C01788=1016.135,48.683,-123.582,-24.251,21.472,-42.282
C01789=1016.137,48.283,-123.546,-24.251,21.474,-42.286
C01790=1016.140,47.883,-123.510,-24.251,21.474,-42.290
C01791=1016.142,47.483,-123.475,-24.250,21.474,-42.295
C01792=1016.145,47.083,-123.439,-24.249,21.475,-42.299
C01793=1016.149,46.682,-123.404,-24.249,21.475,-42.302
C01794=1016.151,46.283,-123.368,-24.248,21.475,-42.308
C01795=1016.153,45.882,-123.332,-24.247,21.475,-42.311
C01796=1016.156,45.482,-123.297,-24.247,21.477,-42.316
C01797=1016.158,45.082,-123.261,-24.246,21.477,-42.321
C01798=1016.161,44.683,-123.225,-24.246,21.477,-42.325
C01799=1016.163,44.282,-123.190,-24.245,21.477,-42.330
C01800=1016.166,43.882,-123.154,-24.244,21.477,-42.333
C01801=1016.169,43.482,-123.119,-24.244,21.479,-42.338
C01802=1016.171,43.082,-123.084,-24.243,21.479,-42.343
C01803=1016.174,42.683,-123.048,-24.243,21.479,-42.347
C01804=1016.177,42.282,-123.012,-24.242,21.479,-42.352
C01805=1016.179,41.882,-122.977,-24.241,21.479,-42.356
C01806=1016.181,41.482,-122.941,-24.241,21.480,-42.359
C01807=1016.184,41.082,-122.906,-24.240,21.481,-42.365
C01808=1016.186,40.683,-122.871,-24.240,21.481,-42.369
C01809=1016.188,40.283,-122.835,-24.239,21.481,-42.374
C01810=1016.191,39.882,-122.800,-24.238,21.481,-42.378
C01811=1016.194,39.483,-122.764,-24.238,21.482,-42.383
C01812=1016.196,39.083,-122.728,-24.237,21.483,-42.387
C01813=1016.199,38.683,-122.694,-24.237,21.483,-42.391
C01814=1016.201,38.283,-122.658,-24.236,21.483,-42.396
C01815=1016.203,37.882,-122.623,-24.235,21.483,-42.400
C01816=1016.205,37.483,-122.587,-24.235,21.484,-42.405
C01817=1016.207,37.084,-122.553,-24.234,21.485,-42.409
C01818=1016.209,36.684,-122.518,-24.233,21.484,-42.414
C01819=1016.212,36.284,-122.482,-24.233,21.485,-42.418
C01820=1016.214,35.884,-122.447,-24.232,21.486,-42.424
C01821=1016.216,35.484,-122.411,-24.231,21.486,-42.428
C01822=1016.219,35.084,-122.376,-24.231,21.486,-42.433
C01823=1016.220,34.685,-122.341,-24.230,21.486,-42.437
C01824=1016.222,34.285,-122.305,-24.229,21.487,-42.442
C01825=1016.225,33.885,-122.271,-24.229,21.488,-42.446
C01826=1016.227,33.486,-122.236,-24.228,21.487,-42.451
C01827=1016.229,33.086,-122.200,-24.228,21.489,-42.455
C01828=1016.232,32.686,-122.165,-24.227,21.489,-42.461
C01829=1016.233,32.287,-122.130,-24.226,21.489,-42.464
C01830=1016.235,31.887,-122.095,-24.226,21.489,-42.469
C01831=1016.237,31.487,-122.060,-24.225,21.490,-42.474
C01832=1016.239,31.087,-122.025,-24.224,21.490,-42.479
C01833=1016.241,30.688,-121.990,-24.224,21.491,-42.483
C01834=1016.243,30.289,-121.954,-24.223,21.491,-42.488
C01835=1016.245,29.889,-121.920,-24.223,21.492,-42.492
C01836=1016.247,29.490,-121.885,-24.222,21.492,-42.497
C01837=1016.249,29.090,-121.850,-24.221,21.492,-42.501
C01838=1016.250,28.691,-121.815,-24.221,21.493,-42.507
C01839=1016.252,28.291,-121.781,-24.220,21.493,-42.510
C01840=1016.255,27.891,-121.745,-24.219,21.493,-42.516
C01841=1016.256,27.492,-121.710,-24.219,21.495,-42.520
C01842=1016.258,27.093,-121.675,-24.218,21.494,-42.525
C01843=1016.260,26.693,-121.641,-24.218,21.495,-42.529
C01844=1016.261,26.294,-121.606,-24.217,21.496,-42.534
C01845=1016.263,25.895,-121.571,-24.216,21.496,-42.540
C01846=1016.265,25.495,-121.536,-24.215,21.496,-42.543
C01847=1016.267,25.096,-121.501,-24.215,21.497,-42.549
C01848=1016.269,24.697,-121.467,-24.214,21.497,-42.553
C01849=1016.271,24.298,-121.432,-24.213,21.497,-42.558
C01850=1016.272,23.915,-121.398,-24.213,21.498,-42.562
C01851=1016.273,23.584,-121.370,-24.213,21.498,-42.564
C01852=1016.275,23.313,-121.346,-24.212,21.498,-42.567
C01853=1016.275,23.078,-121.326,-24.211,21.499,-42.573
C01854=1016.277,22.846,-121.305,-24.211,21.500,-42.577
C01855=1016.278,22.580,-121.283,-24.211,21.500,-42.580
C01856=1016.278,22.258,-121.254,-24.210,21.500,-42.584
C01857=1016.280,21.883,-121.222,-24.210,21.501,-42.586
C01858=1016.282,21.470,-121.186,-24.209,21.501,-42.593
C01859=1016.283,21.225,-121.165,-24.208,21.501,-42.597
C01860=1016.284,20.953,-121.142,-24.208,21.502,-42.599
C01861=1016.285,20.662,-121.116,-24.207,21.501,-42.602
C01862=1016.286,20.365,-121.090,-24.207,21.501,-42.604
C01863=1016.288,20.078,-121.065,-24.207,21.503,-42.606
C01864=1016.288,19.812,-121.042,-24.206,21.502,-42.610
C01865=1016.289,19.575,-121.022,-24.206,21.503,-42.613
C01866=1016.290,19.364,-121.004,-24.205,21.503,-42.617
C01867=1016.291,18.968,-120.970,-24.205,21.503,-42.622
C01868=1016.293,18.571,-120.935,-24.204,21.503,-42.626
C01869=1016.294,18.175,-120.901,-24.203,21.504,-42.632
C01870=1016.296,17.780,-120.867,-24.203,21.505,-42.635
C01871=1016.297,17.386,-120.832,-24.202,21.505,-42.641
C01872=1016.298,16.993,-120.799,-24.201,21.505,-42.646
C01873=1016.299,16.600,-120.765,-24.201,21.506,-42.650
C01874=1016.301,16.208,-120.731,-24.200,21.506,-42.656
C01875=1016.302,15.816,-120.697,-24.200,21.507,-42.659
C01876=1016.304,15.427,-120.664,-24.199,21.507,-42.665
C01877=1016.305,15.037,-120.630,-24.198,21.508,-42.670
C01878=1016.306,14.649,-120.597,-24.198,21.508,-42.674
C01879=1016.307,14.260,-120.563,-24.197,21.509,-42.680
C01880=1016.309,13.873,-120.530,-24.196,21.509,-42.683
C01881=1016.310,13.485,-120.497,-24.196,21.509,-42.689
C01882=1016.311,13.098,-120.463,-24.195,21.511,-42.693
C01883=1016.312,12.712,-120.430,-24.194,21.510,-42.698
C01884=1016.313,12.325,-120.397,-24.193,21.510,-42.703
C01885=1016.314,11.939,-120.364,-24.193,21.512,-42.707
C01886=1016.315,11.552,-120.330,-24.192,21.511,-42.713
C01887=1016.317,11.167,-120.298,-24.192,21.512,-42.716
C01888=1016.317,10.784,-120.265,-24.191,21.513,-42.722
C01889=1016.319,10.403,-120.232,-24.191,21.513,-42.726
C01890=1016.320,10.025,-120.201,-24.190,21.513,-42.731
C01891=1016.320,9.648,-120.168,-24.189,21.514,-42.737
C01892=1016.321,9.273,-120.136,-24.189,21.514,-42.740
C01893=1016.323,8.896,-120.104,-24.188,21.515,-42.746
C01894=1016.323,8.518,-120.071,-24.187,21.515,-42.751
C01895=1016.324,8.138,-120.039,-24.187,21.516,-42.755
C01896=1016.325,7.753,-120.006,-24.186,21.516,-42.761
C01897=1016.327,7.366,-119.973,-24.185,21.517,-42.764
C01898=1016.326,6.975,-119.940,-24.185,21.517,-42.770
C01899=1016.328,6.583,-119.906,-24.184,21.517,-42.775
C01900=1016.329,6.190,-119.873,-24.183,21.519,-42.779
C01901=1016.329,5.797,-119.840,-24.182,21.518,-42.785
C01902=1016.331,5.401,-119.806,-24.182,21.519,-42.790
C01903=1016.331,5.006,-119.772,-24.181,21.520,-42.794
C01904=1016.332,4.612,-119.739,-24.180,21.519,-42.799
C01905=1016.333,4.215,-119.705,-24.180,21.520,-42.805
C01906=1016.333,3.826,-119.672,-24.179,21.521,-42.809
C01907=1016.334,3.467,-119.641,-24.179,21.521,-42.812
C01908=1016.335,3.139,-119.613,-24.178,21.521,-42.817
C01909=1016.335,2.825,-119.586,-24.177,21.522,-42.823
C01910=1016.336,2.503,-119.560,-24.177,21.522,-42.827
C01911=1016.337,2.150,-119.530,-24.176,21.523,-42.833
C01912=1016.337,1.764,-119.496,-24.175,21.524,-42.836
C01913=1016.338,1.367,-119.463,-24.175,21.523,-42.841
C01914=1016.338,0.967,-119.430,-24.174,21.525,-42.846
C01915=1016.339,0.567,-119.396,-24.173,21.525,-42.851
C01916=1016.340,0.166,-119.361,-24.173,21.525,-42.857
C01917=1016.340,-0.237,-119.327,-24.172,21.525,-42.862
C01918=1016.341,-0.644,-119.293,-24.171,21.526,-42.867
C01919=1016.341,-1.051,-119.259,-24.171,21.527,-42.872
C01920=1016.342,-1.462,-119.224,-24.170,21.527,-42.877
C01921=1016.342,-1.874,-119.190,-24.169,21.528,-42.882
C01922=1016.343,-2.289,-119.155,-24.169,21.529,-42.888
C01923=1016.343,-2.705,-119.120,-24.168,21.529,-42.893
C01924=1016.344,-3.125,-119.084,-24.167,21.529,-42.899
C01925=1016.345,-3.547,-119.049,-24.166,21.530,-42.904
C01926=1016.345,-3.758,-119.031,-24.166,21.530,-42.908
C01927=1016.345,-3.970,-119.013,-24.165,21.530,-42.910
C01928=1016.345,-4.184,-118.995,-24.165,21.530,-42.913
C01929=1016.345,-4.400,-118.977,-24.165,21.531,-42.915
C01930=1016.346,-4.616,-118.959,-24.164,21.531,-42.919
C01931=1016.347,-4.834,-118.941,-24.164,21.531,-42.921
C01932=1016.346,-5.054,-118.922,-24.163,21.532,-42.925
C01933=1016.346,-5.276,-118.903,-24.163,21.532,-42.927
C01934=1016.347,-5.499,-118.885,-24.163,21.532,-42.930
C01935=1016.347,-5.722,-118.866,-24.162,21.532,-42.934
C01936=1016.347,-5.946,-118.847,-24.162,21.533,-42.935
C01937=1016.347,-6.171,-118.828,-24.161,21.533,-42.939
C01938=1016.347,-6.394,-118.809,-24.161,21.533,-42.941
C01939=1016.347,-6.618,-118.791,-24.161,21.533,-42.944
C01940=1016.348,-6.842,-118.772,-24.160,21.534,-42.947
C01941=1016.348,-7.064,-118.754,-24.160,21.534,-42.950
C01942=1016.348,-7.285,-118.735,-24.160,21.535,-42.952
C01943=1016.348,-7.506,-118.716,-24.159,21.534,-42.956
C01944=1016.348,-7.725,-118.699,-24.159,21.535,-42.959
C01945=1016.349,-7.943,-118.680,-24.158,21.535,-42.961
C01946=1016.348,-8.160,-118.662,-24.158,21.536,-42.965
C01947=1016.349,-8.377,-118.644,-24.158,21.536,-42.967
C01948=1016.349,-8.594,-118.626,-24.157,21.536,-42.971
C01949=1016.348,-8.810,-118.607,-24.157,21.537,-42.973
C01950=1016.348,-9.027,-118.589,-24.156,21.536,-42.976
C01951=1016.349,-9.243,-118.572,-24.156,21.537,-42.980
C01952=1016.349,-9.460,-118.553,-24.156,21.537,-42.982
C01953=1016.349,-9.676,-118.535,-24.155,21.538,-42.985
C01954=1016.349,-9.893,-118.517,-24.155,21.538,-42.987
C01955=1016.349,-10.108,-118.499,-24.154,21.538,-42.991
C01956=1016.349,-10.324,-118.482,-24.154,21.539,-42.993
C01957=1016.349,-10.539,-118.463,-24.154,21.538,-42.996
C01958=1016.350,-10.754,-118.445,-24.153,21.539,-42.998
C01959=1016.349,-10.969,-118.428,-24.153,21.539,-43.002
C01960=1016.349,-11.183,-118.410,-24.152,21.539,-43.006
C01961=1016.349,-11.396,-118.392,-24.152,21.540,-43.007
C01962=1016.349,-11.610,-118.374,-24.152,21.540,-43.011
C01963=1016.350,-11.822,-118.357,-24.151,21.540,-43.013
C01964=1016.350,-12.035,-118.339,-24.151,21.540,-43.016
C01965=1016.350,-12.247,-118.321,-24.151,21.541,-43.019
C01966=1016.349,-12.458,-118.304,-24.150,21.541,-43.022
C01967=1016.349,-12.670,-118.286,-24.150,21.542,-43.024
C01968=1016.349,-13.089,-118.252,-24.149,21.542,-43.029
C01969=1016.349,-13.506,-118.216,-24.148,21.543,-43.035
C01970=1016.349,-13.921,-118.182,-24.148,21.543,-43.041
C01971=1016.349,-14.332,-118.149,-24.147,21.544,-43.046
C01972=1016.349,-14.741,-118.115,-24.146,21.544,-43.052
C01973=1016.349,-15.146,-118.081,-24.145,21.545,-43.057
C01974=1016.349,-15.549,-118.048,-24.145,21.545,-43.063
C01975=1016.349,-15.950,-118.015,-24.144,21.546,-43.068
C01976=1016.349,-16.349,-117.982,-24.143,21.546,-43.074
C01977=1016.348,-16.748,-117.948,-24.142,21.547,-43.079
C01978=1016.348,-17.146,-117.915,-24.142,21.548,-43.085
C01979=1016.348,-17.544,-117.883,-24.141,21.547,-43.090
C01980=1016.348,-17.955,-117.849,-24.140,21.548,-43.098
C01981=1016.347,-18.203,-117.829,-24.139,21.549,-43.101
C01982=1016.347,-18.490,-117.804,-24.139,21.549,-43.105
C01983=1016.347,-18.802,-117.779,-24.139,21.550,-43.107
C01984=1016.347,-19.113,-117.753,-24.139,21.550,-43.109
C01985=1016.347,-19.401,-117.730,-24.138,21.550,-43.113
C01986=1016.347,-19.651,-117.709,-24.138,21.551,-43.116
C01987=1016.346,-20.061,-117.675,-24.136,21.551,-43.123
C01988=1016.346,-20.459,-117.643,-24.136,21.552,-43.129
C01989=1016.345,-20.857,-117.609,-24.135,21.553,-43.135
C01990=1016.345,-21.254,-117.577,-24.134,21.552,-43.140
C01991=1016.345,-21.652,-117.544,-24.134,21.553,-43.146
C01992=1016.344,-22.049,-117.512,-24.133,21.554,-43.151
C01993=1016.344,-22.447,-117.479,-24.132,21.554,-43.156
C01994=1016.343,-22.844,-117.447,-24.131,21.555,-43.162
C01995=1016.342,-23.242,-117.414,-24.131,21.555,-43.168
C01996=1016.342,-23.639,-117.382,-24.130,21.556,-43.173
C01997=1016.342,-24.037,-117.349,-24.129,21.556,-43.178
C01998=1016.341,-24.434,-117.317,-24.128,21.557,-43.184
C01999=1016.341,-24.832,-117.284,-24.128,21.558,-43.190
C02000=1016.340,-25.229,-117.252,-24.127,21.558,-43.195
C02001=1016.339,-25.627,-117.219,-24.126,21.558,-43.201
C02002=1016.339,-26.024,-117.187,-24.125,21.559,-43.206
C02003=1016.338,-26.422,-117.154,-24.125,21.560,-43.212
C02004=1016.337,-26.819,-117.122,-24.124,21.560,-43.217
C02005=1016.336,-27.216,-117.090,-24.123,21.561,-43.221
C02006=1016.336,-27.614,-117.057,-24.123,21.562,-43.227
C02007=1016.335,-28.012,-117.025,-24.122,21.562,-43.232
C02008=1016.334,-28.410,-116.993,-24.121,21.562,-43.238
C02009=1016.334,-28.807,-116.961,-24.120,21.563,-43.243
C02010=1016.333,-29.204,-116.929,-24.120,21.564,-43.249
C02011=1016.331,-29.602,-116.896,-24.119,21.565,-43.255
C02012=1016.331,-29.999,-116.864,-24.118,21.565,-43.260
C02013=1016.330,-30.397,-116.832,-24.117,21.565,-43.265
C02014=1016.329,-30.794,-116.800,-24.117,21.566,-43.271
C02015=1016.328,-31.191,-116.768,-24.116,21.567,-43.277
C02016=1016.327,-31.589,-116.735,-24.115,21.568,-43.282
C02017=1016.326,-31.986,-116.703,-24.114,21.567,-43.287
C02018=1016.325,-32.383,-116.671,-24.114,21.568,-43.293
C02019=1016.325,-32.781,-116.639,-24.113,21.569,-43.299
C02020=1016.323,-33.179,-116.607,-24.112,21.570,-43.304
C02021=1016.322,-33.576,-116.575,-24.111,21.570,-43.310
C02022=1016.321,-33.973,-116.543,-24.111,21.570,-43.315
C02023=1016.321,-34.371,-116.511,-24.110,21.571,-43.321
C02024=1016.319,-34.768,-116.479,-24.109,21.571,-43.328
C02025=1016.318,-35.166,-116.447,-24.108,21.572,-43.334
C02026=1016.317,-35.563,-116.414,-24.107,21.572,-43.339
C02027=1016.315,-35.960,-116.383,-24.107,21.573,-43.344
C02028=1016.315,-36.357,-116.351,-24.106,21.573,-43.350
C02029=1016.313,-36.755,-116.319,-24.105,21.574,-43.356
C02030=1016.312,-37.152,-116.287,-24.105,21.575,-43.361
C02031=1016.311,-37.549,-116.256,-24.104,21.575,-43.366
C02032=1016.310,-37.947,-116.223,-24.103,21.576,-43.372
C02033=1016.308,-38.344,-116.192,-24.102,21.576,-43.378
C02034=1016.307,-38.741,-116.159,-24.102,21.577,-43.383
C02035=1016.305,-39.138,-116.128,-24.101,21.578,-43.389
C02036=1016.304,-39.536,-116.097,-24.100,21.578,-43.394
C02037=1016.303,-39.934,-116.064,-24.099,21.579,-43.400
C02038=1016.301,-40.331,-116.033,-24.099,21.579,-43.405
C02039=1016.300,-40.728,-116.001,-24.098,21.580,-43.411
C02040=1016.298,-41.126,-115.969,-24.097,21.581,-43.417
C02041=1016.297,-41.523,-115.937,-24.096,21.582,-43.422
C02042=1016.296,-41.920,-115.906,-24.096,21.582,-43.427
C02043=1016.294,-42.317,-115.875,-24.095,21.582,-43.433
C02044=1016.292,-42.715,-115.843,-24.094,21.583,-43.439
C02045=1016.291,-43.112,-115.811,-24.093,21.584,-43.444
C02046=1016.289,-43.509,-115.779,-24.092,21.584,-43.451
C02047=1016.288,-43.906,-115.749,-24.092,21.585,-43.457
C02048=1016.286,-44.304,-115.717,-24.091,21.585,-43.462
C02049=1016.284,-44.701,-115.685,-24.090,21.585,-43.468
C02050=1016.283,-45.098,-115.653,-24.089,21.586,-43.473
C02051=1016.281,-45.495,-115.622,-24.089,21.587,-43.479
C02052=1016.279,-45.892,-115.590,-24.088,21.588,-43.485
C02053=1016.278,-46.290,-115.559,-24.087,21.589,-43.490
C02054=1016.276,-46.687,-115.527,-24.086,21.588,-43.496
C02055=1016.274,-47.083,-115.496,-24.086,21.589,-43.501
C02056=1016.272,-47.481,-115.464,-24.085,21.590,-43.507
C02057=1016.271,-47.878,-115.433,-24.084,21.591,-43.512
C02058=1016.269,-48.275,-115.402,-24.084,21.592,-43.518
C02059=1016.267,-48.673,-115.371,-24.083,21.592,-43.525
C02060=1016.265,-49.070,-115.339,-24.082,21.592,-43.531
C02061=1016.263,-49.466,-115.308,-24.081,21.592,-43.536
C02062=1016.261,-49.863,-115.276,-24.080,21.593,-43.542
C02063=1016.259,-50.261,-115.244,-24.080,21.594,-43.547
C02064=1016.257,-50.658,-115.214,-24.079,21.595,-43.553
C02065=1016.255,-51.055,-115.183,-24.078,21.595,-43.558
C02066=1016.253,-51.452,-115.152,-24.077,21.596,-43.564
C02067=1016.251,-51.848,-115.121,-24.077,21.597,-43.570
C02068=1016.249,-52.246,-115.089,-24.076,21.598,-43.575
C02069=1016.247,-52.642,-115.058,-24.075,21.598,-43.581
C02070=1016.245,-53.039,-115.027,-24.074,21.598,-43.588
C02071=1016.242,-53.436,-114.996,-24.073,21.599,-43.593
C02072=1016.241,-53.833,-114.965,-24.073,21.599,-43.599
C02073=1016.238,-54.231,-114.933,-24.072,21.600,-43.604
C02074=1016.236,-54.627,-114.902,-24.071,21.601,-43.610
C02075=1016.234,-55.024,-114.871,-24.071,21.602,-43.616
C02076=1016.231,-55.421,-114.840,-24.070,21.603,-43.621
C02077=1016.230,-55.819,-114.809,-24.069,21.602,-43.627
C02078=1016.227,-56.216,-114.778,-24.068,21.603,-43.632
C02079=1016.224,-56.614,-114.747,-24.067,21.603,-43.639
C02080=1016.223,-57.012,-114.716,-24.067,21.604,-43.645
C02081=1016.220,-57.410,-114.685,-24.066,21.605,-43.651
C02082=1016.218,-57.809,-114.654,-24.065,21.606,-43.656
C02083=1016.215,-58.208,-114.623,-24.064,21.606,-43.662
C02084=1016.212,-58.607,-114.592,-24.064,21.607,-43.667
C02085=1016.210,-59.008,-114.561,-24.063,21.608,-43.673
C02086=1016.208,-59.409,-114.529,-24.062,21.608,-43.680
C02087=1016.205,-59.811,-114.499,-24.061,21.609,-43.686
C02088=1016.202,-60.212,-114.468,-24.061,21.610,-43.691
C02089=1016.200,-60.614,-114.436,-24.060,21.610,-43.697
C02090=1016.197,-61.018,-114.405,-24.059,21.610,-43.702
C02091=1016.195,-61.421,-114.374,-24.058,21.611,-43.708
C02092=1016.192,-61.825,-114.342,-24.057,21.611,-43.715
C02093=1016.190,-62.230,-114.311,-24.057,21.612,-43.720
C02094=1016.186,-62.635,-114.280,-24.056,21.613,-43.726
C02095=1016.183,-63.041,-114.248,-24.055,21.614,-43.732
C02096=1016.181,-63.447,-114.217,-24.054,21.615,-43.737
C02097=1016.178,-63.854,-114.185,-24.053,21.615,-43.744
C02098=1016.175,-64.261,-114.154,-24.053,21.615,-43.750
C02099=1016.171,-64.669,-114.122,-24.052,21.616,-43.756
C02100=1016.170,-65.077,-114.091,-24.051,21.617,-43.761
C02101=1016.166,-65.486,-114.060,-24.050,21.617,-43.768
C02102=1016.163,-65.895,-114.028,-24.049,21.618,-43.774
C02103=1016.161,-66.303,-113.996,-24.049,21.619,-43.780
C02104=1016.157,-66.713,-113.965,-24.048,21.620,-43.785
C02105=1016.154,-67.122,-113.933,-24.047,21.620,-43.791
C02106=1016.151,-67.533,-113.902,-24.046,21.621,-43.798
C02107=1016.148,-67.943,-113.870,-24.046,21.621,-43.804
C02108=1016.144,-68.354,-113.839,-24.045,21.622,-43.809
C02109=1016.141,-68.764,-113.807,-24.044,21.623,-43.815
C02110=1016.138,-69.175,-113.776,-24.043,21.623,-43.822
C02111=1016.135,-69.585,-113.744,-24.042,21.624,-43.827
C02112=1016.131,-69.997,-113.713,-24.042,21.625,-43.833
C02113=1016.128,-70.407,-113.681,-24.041,21.625,-43.839
C02114=1016.125,-70.818,-113.650,-24.040,21.626,-43.846
C02115=1016.122,-71.229,-113.619,-24.039,21.626,-43.851
C02116=1016.118,-71.640,-113.587,-24.039,21.627,-43.857
C02117=1016.115,-72.052,-113.556,-24.038,21.628,-43.865
C02118=1016.112,-72.462,-113.524,-24.037,21.629,-43.870
C02119=1016.107,-72.873,-113.493,-24.036,21.630,-43.876
C02120=1016.104,-73.283,-113.462,-24.035,21.631,-43.881
C02121=1016.101,-73.695,-113.431,-24.034,21.631,-43.888
C02122=1016.097,-74.105,-113.399,-24.034,21.632,-43.894
C02123=1016.093,-74.516,-113.368,-24.033,21.632,-43.900
C02124=1016.089,-74.926,-113.337,-24.032,21.633,-43.905
C02125=1016.086,-75.336,-113.305,-24.031,21.633,-43.912
C02126=1016.083,-75.746,-113.275,-24.031,21.634,-43.918
C02127=1016.078,-76.156,-113.243,-24.030,21.635,-43.924
C02128=1016.075,-76.565,-113.212,-24.029,21.636,-43.929
C02129=1016.071,-76.974,-113.181,-24.028,21.636,-43.936
C02130=1016.068,-77.383,-113.150,-24.027,21.637,-43.942
C02131=1016.064,-77.791,-113.119,-24.027,21.637,-43.948
C02132=1016.060,-78.199,-113.088,-24.026,21.638,-43.953
C02133=1016.056,-78.607,-113.057,-24.025,21.638,-43.960
C02134=1016.052,-79.014,-113.026,-24.024,21.639,-43.966
C02135=1016.048,-79.421,-112.995,-24.023,21.640,-43.972
C02136=1016.044,-79.826,-112.965,-24.023,21.641,-43.977
C02137=1016.040,-80.233,-112.934,-24.022,21.641,-43.984
C02138=1016.036,-80.638,-112.904,-24.021,21.642,-43.990
C02139=1016.032,-81.042,-112.873,-24.020,21.643,-43.995
C02140=1016.028,-81.446,-112.843,-24.020,21.643,-44.001
C02141=1016.024,-81.850,-112.812,-24.019,21.644,-44.007
C02142=1016.020,-82.252,-112.782,-24.018,21.644,-44.014
C02143=1016.016,-82.654,-112.752,-24.017,21.645,-44.019
C02144=1016.012,-83.056,-112.721,-24.016,21.646,-44.025
C02145=1016.008,-83.457,-112.692,-24.016,21.647,-44.031
C02146=1016.003,-83.857,-112.661,-24.015,21.648,-44.036
C02147=1015.999,-84.257,-112.631,-24.014,21.648,-44.043
C02148=1015.995,-84.663,-112.600,-24.013,21.649,-44.049
C02149=1015.992,-84.887,-112.584,-24.013,21.649,-44.053
C02150=1015.989,-85.128,-112.566,-24.012,21.650,-44.056
C02151=1015.988,-85.381,-112.547,-24.012,21.649,-44.060
C02152=1015.984,-85.636,-112.528,-24.012,21.650,-44.062
C02153=1015.981,-85.882,-112.509,-24.011,21.650,-44.065
C02154=1015.979,-86.111,-112.492,-24.011,21.651,-44.069
C02155=1015.974,-86.522,-112.461,-24.010,21.652,-44.077
C02156=1015.970,-86.909,-112.432,-24.009,21.652,-44.082
C02157=1015.967,-87.289,-112.403,-24.008,21.652,-44.087
C02158=1015.962,-87.661,-112.375,-24.007,21.653,-44.093
C02159=1015.958,-88.033,-112.347,-24.007,21.654,-44.099
C02160=1015.953,-88.409,-112.320,-24.006,21.655,-44.104
C02161=1015.949,-88.816,-112.289,-24.005,21.656,-44.112
C02162=1015.946,-89.063,-112.271,-24.005,21.656,-44.116
C02163=1015.943,-89.339,-112.250,-24.004,21.657,-44.117
C02164=1015.940,-89.623,-112.229,-24.004,21.656,-44.121
C02165=1015.936,-89.897,-112.209,-24.003,21.657,-44.124
C02166=1015.933,-90.148,-112.190,-24.003,21.657,-44.128
C02167=1015.931,-90.366,-112.173,-24.002,21.658,-44.132
C02168=1015.926,-90.762,-112.144,-24.002,21.659,-44.138
C02169=1015.921,-91.156,-112.115,-24.001,21.659,-44.145
C02170=1015.917,-91.548,-112.086,-24.000,21.660,-44.150
C02171=1015.912,-91.941,-112.056,-23.999,21.660,-44.156
C02172=1015.908,-92.332,-112.027,-23.999,21.661,-44.162
C02173=1015.903,-92.723,-111.998,-23.998,21.662,-44.167
C02174=1015.898,-93.113,-111.968,-23.997,21.663,-44.173
C02175=1015.893,-93.502,-111.940,-23.996,21.664,-44.178
C02176=1015.888,-93.890,-111.911,-23.996,21.664,-44.184
C02177=1015.883,-94.278,-111.882,-23.995,21.664,-44.189
C02178=1015.879,-94.665,-111.854,-23.994,21.665,-44.195
C02179=1015.873,-95.051,-111.825,-23.994,21.666,-44.200
C02180=1015.869,-95.437,-111.796,-23.993,21.666,-44.207
C02181=1015.864,-95.822,-111.767,-23.992,21.667,-44.213
C02182=1015.859,-96.206,-111.739,-23.991,21.668,-44.219
C02183=1015.854,-96.591,-111.710,-23.990,21.668,-44.224
C02184=1015.848,-96.975,-111.682,-23.990,21.669,-44.230
C02185=1015.843,-97.358,-111.654,-23.989,21.669,-44.235
C02186=1015.839,-97.742,-111.625,-23.988,21.670,-44.241
C02187=1015.833,-98.125,-111.596,-23.988,21.671,-44.246
C02188=1015.829,-98.508,-111.568,-23.987,21.672,-44.252
C02189=1015.824,-98.891,-111.541,-23.986,21.673,-44.258
C02190=1015.818,-99.275,-111.512,-23.985,21.673,-44.263
C02191=1015.812,-99.659,-111.483,-23.985,21.673,-44.268
C02192=1015.807,-100.043,-111.454,-23.984,21.674,-44.274
C02193=1015.802,-100.428,-111.427,-23.983,21.675,-44.280
C02194=1015.797,-100.813,-111.398,-23.982,21.676,-44.285
C02195=1015.791,-101.199,-111.370,-23.982,21.677,-44.291
C02196=1015.786,-101.585,-111.341,-23.981,21.676,-44.296
C02197=1015.780,-101.972,-111.313,-23.980,21.677,-44.302
C02198=1015.775,-102.360,-111.284,-23.980,21.678,-44.307
C02199=1015.769,-102.748,-111.256,-23.979,21.678,-44.314
C02200=1015.764,-103.138,-111.227,-23.978,21.679,-44.320
C02201=1015.758,-103.527,-111.198,-23.977,21.680,-44.326
C02202=1015.753,-103.918,-111.170,-23.976,21.681,-44.331
C02203=1015.747,-104.310,-111.141,-23.976,21.682,-44.337
C02204=1015.741,-104.701,-111.112,-23.975,21.681,-44.342
C02205=1015.735,-105.093,-111.083,-23.974,21.682,-44.348
C02206=1015.730,-105.486,-111.054,-23.974,21.683,-44.353
C02207=1015.723,-105.878,-111.026,-23.973,21.684,-44.359
C02208=1015.718,-106.271,-110.997,-23.972,21.685,-44.365
C02209=1015.712,-106.664,-110.968,-23.971,21.686,-44.370
C02210=1015.706,-107.057,-110.939,-23.971,21.686,-44.376
C02211=1015.700,-107.450,-110.910,-23.970,21.687,-44.383
C02212=1015.693,-107.843,-110.881,-23.969,21.687,-44.388
C02213=1015.687,-108.236,-110.852,-23.968,21.688,-44.394
C02214=1015.681,-108.629,-110.823,-23.968,21.688,-44.399
C02215=1015.675,-109.022,-110.795,-23.967,21.689,-44.405
C02216=1015.669,-109.415,-110.766,-23.966,21.690,-44.411
C02217=1015.663,-109.808,-110.737,-23.965,21.691,-44.416
C02218=1015.656,-110.201,-110.709,-23.965,21.691,-44.422
C02219=1015.650,-110.594,-110.680,-23.964,21.692,-44.427
C02220=1015.644,-110.987,-110.651,-23.963,21.693,-44.433
C02221=1015.637,-111.380,-110.623,-23.963,21.694,-44.439
C02222=1015.631,-111.772,-110.593,-23.962,21.694,-44.446
C02223=1015.624,-112.164,-110.565,-23.961,21.694,-44.451
C02224=1015.618,-112.557,-110.536,-23.960,21.695,-44.456
C02225=1015.611,-112.950,-110.508,-23.959,21.696,-44.462
C02226=1015.605,-113.343,-110.479,-23.959,21.696,-44.468
C02227=1015.598,-113.735,-110.450,-23.958,21.697,-44.473
C02228=1015.592,-114.128,-110.422,-23.957,21.698,-44.479
C02229=1015.585,-114.520,-110.392,-23.957,21.699,-44.485
C02230=1015.578,-114.913,-110.364,-23.956,21.700,-44.490
C02231=1015.571,-115.306,-110.335,-23.955,21.701,-44.496
C02232=1015.565,-115.699,-110.307,-23.954,21.700,-44.501
C02233=1015.557,-116.090,-110.278,-23.954,21.701,-44.507
C02234=1015.550,-116.483,-110.250,-23.953,21.702,-44.512
C02235=1015.543,-116.876,-110.221,-23.952,21.703,-44.518
C02236=1015.536,-117.268,-110.192,-23.952,21.704,-44.523
C02237=1015.530,-117.661,-110.164,-23.951,21.705,-44.529
C02238=1015.522,-118.053,-110.136,-23.950,21.705,-44.536
C02239=1015.515,-118.445,-110.107,-23.949,21.705,-44.541
C02240=1015.508,-118.838,-110.079,-23.948,21.706,-44.547
C02241=1015.501,-119.230,-110.050,-23.948,21.706,-44.553
C02242=1015.494,-119.623,-110.021,-23.947,21.707,-44.558
C02243=1015.487,-120.015,-109.993,-23.946,21.708,-44.564
C02244=1015.479,-120.407,-109.965,-23.946,21.709,-44.569
C02245=1015.472,-120.800,-109.936,-23.945,21.710,-44.575
C02246=1015.465,-121.191,-109.907,-23.944,21.710,-44.580
C02247=1015.457,-121.583,-109.879,-23.943,21.710,-44.586
C02248=1015.452,-121.872,-109.858,-23.943,21.711,-44.590
C02249=1015.446,-122.160,-109.837,-23.943,21.712,-44.594
C02250=1015.442,-122.368,-109.822,-23.942,21.712,-44.597
C02251=1015.435,-122.760,-109.794,-23.941,21.713,-44.603
C02252=1015.427,-123.152,-109.765,-23.941,21.714,-44.608
C02253=1015.419,-123.544,-109.737,-23.940,21.715,-44.614
C02254=1015.413,-123.937,-109.708,-23.939,21.714,-44.619
C02255=1015.404,-124.329,-109.679,-23.939,21.715,-44.625
C02256=1015.397,-124.722,-109.651,-23.938,21.716,-44.630
C02257=1015.389,-125.113,-109.623,-23.937,21.717,-44.636
C02258=1015.381,-125.505,-109.595,-23.936,21.718,-44.642
C02259=1015.373,-125.897,-109.566,-23.936,21.719,-44.647
C02260=1015.366,-126.289,-109.538,-23.935,21.719,-44.652
C02261=1015.357,-126.682,-109.509,-23.934,21.719,-44.658
C02262=1015.349,-127.073,-109.481,-23.934,21.720,-44.664
C02263=1015.341,-127.465,-109.453,-23.933,21.721,-44.669
C02264=1015.333,-127.857,-109.424,-23.932,21.722,-44.675
C02265=1015.325,-128.250,-109.396,-23.932,21.723,-44.680
C02266=1015.317,-128.641,-109.368,-23.931,21.723,-44.686
C02267=1015.309,-129.033,-109.339,-23.930,21.723,-44.691
C02268=1015.301,-129.426,-109.310,-23.929,21.724,-44.697
C02269=1015.292,-129.817,-109.282,-23.929,21.725,-44.703
C02270=1015.284,-130.209,-109.254,-23.928,21.726,-44.708
C02271=1015.275,-130.601,-109.225,-23.927,21.727,-44.714
C02272=1015.267,-130.993,-109.197,-23.926,21.727,-44.719
C02273=1015.258,-131.385,-109.168,-23.926,21.728,-44.725
C02274=1015.250,-131.777,-109.140,-23.925,21.728,-44.730
C02275=1015.241,-132.169,-109.112,-23.924,21.729,-44.736
C02276=1015.232,-132.560,-109.084,-23.924,21.730,-44.741
C02277=1015.224,-132.953,-109.055,-23.923,21.730,-44.747
C02278=1015.216,-133.344,-109.027,-23.922,21.731,-44.752
C02279=1015.206,-133.737,-108.998,-23.922,21.732,-44.758
C02280=1015.198,-134.128,-108.970,-23.921,21.732,-44.763
C02281=1015.617,-134.098,-109.231,-23.921,21.732,-44.763
C02282=1015.625,-133.706,-109.260,-23.922,21.732,-44.758
C02283=1015.633,-133.314,-109.287,-23.922,21.731,-44.752
C02284=1015.642,-132.922,-109.316,-23.923,21.730,-44.747
C02285=1015.650,-132.531,-109.344,-23.924,21.730,-44.741
C02286=1015.658,-132.139,-109.372,-23.924,21.729,-44.736
C02287=1015.666,-131.747,-109.400,-23.925,21.728,-44.730
C02288=1015.674,-131.355,-109.428,-23.926,21.728,-44.725
C02289=1015.683,-130.963,-109.456,-23.926,21.727,-44.719
C02290=1015.690,-130.571,-109.484,-23.927,21.727,-44.714
C02291=1015.699,-130.179,-109.512,-23.928,21.726,-44.708
C02292=1015.706,-129.787,-109.540,-23.929,21.725,-44.703
C02293=1015.714,-129.395,-109.569,-23.929,21.724,-44.697
C02294=1015.722,-129.004,-109.597,-23.930,21.723,-44.691
C02295=1015.730,-128.611,-109.625,-23.931,21.723,-44.686
C02296=1015.737,-128.220,-109.653,-23.932,21.723,-44.680
C02297=1015.746,-127.827,-109.680,-23.932,21.722,-44.675
C02298=1015.753,-127.436,-109.709,-23.933,21.721,-44.669
C02299=1015.761,-127.043,-109.737,-23.934,21.720,-44.664
C02300=1015.769,-126.651,-109.766,-23.934,21.719,-44.658
C02301=1015.776,-126.259,-109.793,-23.935,21.719,-44.652
C02302=1015.784,-125.867,-109.822,-23.936,21.719,-44.647
C02303=1015.791,-125.475,-109.850,-23.936,21.718,-44.642
C02304=1015.798,-125.084,-109.878,-23.937,21.717,-44.636
C02305=1015.806,-124.691,-109.906,-23.938,21.716,-44.630
C02306=1015.813,-124.299,-109.935,-23.939,21.715,-44.625
C02307=1015.821,-123.907,-109.963,-23.939,21.714,-44.619
C02308=1015.828,-123.515,-109.992,-23.940,21.715,-44.614
C02309=1015.835,-123.123,-110.019,-23.941,21.714,-44.608
C02310=1015.842,-122.731,-110.047,-23.941,21.713,-44.603
C02311=1015.850,-122.339,-110.076,-23.942,21.712,-44.597
C02312=1015.857,-121.946,-110.104,-23.943,21.711,-44.591
C02313=1015.864,-121.554,-110.132,-23.943,21.710,-44.586
C02314=1015.871,-121.162,-110.161,-23.944,21.710,-44.580
C02315=1015.878,-120.770,-110.189,-23.945,21.710,-44.575
C02316=1015.885,-120.377,-110.217,-23.946,21.709,-44.569
C02317=1015.891,-119.985,-110.245,-23.946,21.708,-44.564
C02318=1015.898,-119.593,-110.274,-23.947,21.707,-44.558
C02319=1015.906,-119.201,-110.302,-23.948,21.706,-44.553
C02320=1015.913,-118.808,-110.331,-23.948,21.706,-44.547
C02321=1015.919,-118.416,-110.359,-23.949,21.705,-44.541
C02322=1015.926,-118.024,-110.387,-23.950,21.705,-44.536
C02323=1015.933,-117.631,-110.416,-23.951,21.705,-44.529
C02324=1015.939,-117.239,-110.444,-23.952,21.704,-44.523
C02325=1015.946,-116.847,-110.472,-23.952,21.703,-44.518
C02326=1015.953,-116.454,-110.501,-23.953,21.702,-44.512
C02327=1015.959,-116.062,-110.529,-23.954,21.701,-44.507
C02328=1015.965,-115.669,-110.557,-23.954,21.700,-44.501
C02329=1015.972,-115.276,-110.586,-23.955,21.701,-44.496
C02330=1015.978,-114.884,-110.614,-23.956,21.700,-44.490
C02331=1015.985,-114.492,-110.643,-23.957,21.699,-44.485
C02332=1015.992,-114.099,-110.671,-23.957,21.698,-44.479
C02333=1015.998,-113.706,-110.700,-23.958,21.697,-44.473
C02334=1016.004,-113.314,-110.728,-23.959,21.696,-44.468
C02335=1016.010,-112.921,-110.757,-23.959,21.696,-44.462
C02336=1016.017,-112.528,-110.785,-23.960,21.695,-44.456
C02337=1016.023,-112.136,-110.813,-23.961,21.694,-44.451
C02338=1016.029,-111.743,-110.842,-23.962,21.694,-44.446
C02339=1016.036,-111.350,-110.871,-23.963,21.694,-44.439
C02340=1016.041,-110.957,-110.899,-23.963,21.693,-44.433
C02341=1016.048,-110.565,-110.927,-23.964,21.692,-44.427
C02342=1016.054,-110.172,-110.957,-23.965,21.691,-44.422
C02343=1016.060,-109.780,-110.985,-23.965,21.691,-44.416
C02344=1016.066,-109.387,-111.014,-23.966,21.690,-44.411
C02345=1016.071,-108.993,-111.042,-23.967,21.689,-44.405
C02346=1016.078,-108.600,-111.071,-23.968,21.688,-44.399
C02347=1016.083,-108.208,-111.099,-23.968,21.688,-44.394
C02348=1016.089,-107.815,-111.128,-23.969,21.687,-44.388
C02349=1016.095,-107.421,-111.157,-23.970,21.687,-44.383
C02350=1016.101,-107.028,-111.186,-23.971,21.686,-44.376
C02351=1016.107,-106.636,-111.214,-23.971,21.686,-44.370
C02352=1016.113,-106.242,-111.242,-23.972,21.685,-44.365
C02353=1016.119,-105.849,-111.271,-23.973,21.684,-44.359
C02354=1016.124,-105.457,-111.300,-23.974,21.683,-44.353
C02355=1016.129,-105.064,-111.329,-23.974,21.682,-44.348
C02356=1016.135,-104.672,-111.358,-23.975,21.681,-44.342
C02357=1016.141,-104.281,-111.386,-23.976,21.682,-44.337
C02358=1016.146,-103.889,-111.415,-23.976,21.681,-44.331
C02359=1016.151,-103.500,-111.444,-23.977,21.680,-44.326
C02360=1016.157,-103.109,-111.472,-23.978,21.679,-44.320
C02361=1016.162,-102.720,-111.501,-23.979,21.678,-44.314
C02362=1016.167,-102.332,-111.529,-23.980,21.678,-44.307
C02363=1016.173,-101.944,-111.558,-23.980,21.677,-44.302
C02364=1016.178,-101.557,-111.586,-23.981,21.676,-44.296
C02365=1016.184,-101.170,-111.614,-23.982,21.677,-44.291
C02366=1016.189,-100.784,-111.642,-23.982,21.676,-44.285
C02367=1016.193,-100.399,-111.671,-23.983,21.675,-44.280
C02368=1016.200,-100.015,-111.699,-23.984,21.674,-44.274
C02369=1016.203,-99.630,-111.727,-23.985,21.673,-44.268
C02370=1016.209,-99.246,-111.755,-23.985,21.673,-44.263
C02371=1016.214,-98.863,-111.783,-23.986,21.673,-44.258
C02372=1016.219,-98.480,-111.811,-23.987,21.672,-44.252
C02373=1016.225,-98.096,-111.840,-23.988,21.671,-44.246
C02374=1016.229,-97.713,-111.869,-23.988,21.670,-44.241
C02375=1016.234,-97.330,-111.897,-23.989,21.669,-44.235
C02376=1016.239,-96.946,-111.925,-23.990,21.669,-44.230
C02377=1016.243,-96.563,-111.953,-23.990,21.668,-44.224
C02378=1016.248,-96.179,-111.982,-23.991,21.668,-44.219
C02379=1016.253,-95.794,-112.010,-23.992,21.667,-44.213
C02380=1016.258,-95.409,-112.039,-23.993,21.666,-44.207
C02381=1016.262,-95.023,-112.067,-23.994,21.666,-44.200
C02382=1016.267,-94.637,-112.096,-23.994,21.665,-44.195
C02383=1016.272,-94.250,-112.124,-23.995,21.664,-44.189
C02384=1016.277,-93.863,-112.153,-23.996,21.664,-44.184
C02385=1016.281,-93.474,-112.182,-23.996,21.664,-44.178
C02386=1016.286,-93.085,-112.210,-23.997,21.663,-44.173
C02387=1016.290,-92.695,-112.239,-23.998,21.662,-44.167
C02388=1016.295,-92.304,-112.268,-23.999,21.661,-44.162
C02389=1016.300,-91.913,-112.298,-23.999,21.660,-44.156
C02390=1016.304,-91.521,-112.327,-24.000,21.660,-44.150
C02391=1016.308,-91.128,-112.356,-24.001,21.659,-44.145
C02392=1016.313,-90.734,-112.385,-24.002,21.659,-44.138
C02393=1016.318,-90.338,-112.414,-24.002,21.658,-44.132
C02394=1016.320,-90.120,-112.430,-24.003,21.657,-44.128
C02395=1016.323,-89.870,-112.450,-24.003,21.657,-44.124
C02396=1016.326,-89.595,-112.470,-24.004,21.656,-44.121
C02397=1016.329,-89.310,-112.491,-24.004,21.657,-44.117
C02398=1016.332,-89.036,-112.511,-24.005,21.656,-44.116
C02399=1016.334,-88.788,-112.530,-24.005,21.656,-44.112
C02400=1016.339,-88.381,-112.560,-24.006,21.655,-44.104
C02401=1016.344,-88.006,-112.589,-24.007,21.654,-44.099
C02402=1016.348,-87.634,-112.616,-24.007,21.653,-44.093
C02403=1016.352,-87.261,-112.644,-24.008,21.652,-44.087
C02404=1016.355,-86.882,-112.672,-24.009,21.652,-44.082
C02405=1016.360,-86.494,-112.702,-24.010,21.652,-44.077
C02406=1016.364,-86.084,-112.732,-24.011,21.651,-44.069
C02407=1016.366,-85.855,-112.749,-24.011,21.650,-44.065
C02408=1016.369,-85.608,-112.767,-24.012,21.650,-44.062
C02409=1016.372,-85.354,-112.786,-24.012,21.649,-44.060
C02410=1016.375,-85.100,-112.806,-24.012,21.650,-44.056
C02411=1016.376,-84.859,-112.823,-24.013,21.649,-44.053
C02412=1016.379,-84.635,-112.840,-24.013,21.649,-44.049
C02413=1016.383,-84.229,-112.870,-24.014,21.648,-44.043
C02414=1016.387,-83.829,-112.900,-24.015,21.648,-44.036
C02415=1016.392,-83.430,-112.931,-24.016,21.647,-44.031
C02416=1016.395,-83.028,-112.961,-24.016,21.646,-44.025
C02417=1016.399,-82.627,-112.991,-24.017,21.645,-44.019
C02418=1016.403,-82.224,-113.021,-24.018,21.644,-44.014
C02419=1016.407,-81.821,-113.051,-24.019,21.644,-44.007
C02420=1016.412,-81.418,-113.081,-24.020,21.643,-44.001
C02421=1016.415,-81.014,-113.112,-24.020,21.643,-43.995
C02422=1016.419,-80.610,-113.143,-24.021,21.642,-43.990
C02423=1016.423,-80.205,-113.173,-24.022,21.641,-43.984
C02424=1016.426,-79.799,-113.204,-24.023,21.641,-43.977
C02425=1016.431,-79.393,-113.234,-24.023,21.640,-43.972
C02426=1016.435,-78.986,-113.265,-24.024,21.639,-43.966
C02427=1016.438,-78.579,-113.295,-24.025,21.638,-43.960
C02428=1016.442,-78.171,-113.326,-24.026,21.638,-43.953
C02429=1016.446,-77.763,-113.358,-24.027,21.637,-43.948
C02430=1016.450,-77.355,-113.388,-24.027,21.637,-43.942
C02431=1016.453,-76.946,-113.419,-24.028,21.636,-43.936
C02432=1016.457,-76.537,-113.450,-24.029,21.636,-43.929
C02433=1016.460,-76.128,-113.481,-24.030,21.635,-43.924
C02434=1016.464,-75.719,-113.512,-24.031,21.634,-43.918
C02435=1016.467,-75.309,-113.544,-24.031,21.633,-43.912
C02436=1016.471,-74.898,-113.575,-24.032,21.633,-43.905
C02437=1016.475,-74.488,-113.605,-24.033,21.632,-43.900
C02438=1016.478,-74.078,-113.637,-24.034,21.632,-43.894
C02439=1016.481,-73.666,-113.668,-24.034,21.631,-43.888
C02440=1016.485,-73.257,-113.699,-24.035,21.631,-43.881
C02441=1016.488,-72.846,-113.730,-24.036,21.630,-43.876
C02442=1016.491,-72.435,-113.761,-24.037,21.629,-43.870
C02443=1016.495,-72.024,-113.793,-24.038,21.628,-43.865
C02444=1016.498,-71.613,-113.824,-24.039,21.627,-43.857
C02445=1016.501,-71.202,-113.856,-24.039,21.626,-43.851
C02446=1016.505,-70.791,-113.887,-24.040,21.626,-43.846
C02447=1016.508,-70.380,-113.918,-24.041,21.625,-43.839
C02448=1016.511,-69.969,-113.950,-24.042,21.625,-43.833
C02449=1016.514,-69.558,-113.981,-24.042,21.624,-43.827
C02450=1016.518,-69.147,-114.013,-24.043,21.623,-43.822
C02451=1016.521,-68.737,-114.044,-24.044,21.623,-43.815
C02452=1016.524,-68.326,-114.076,-24.045,21.622,-43.809
C02453=1016.526,-67.916,-114.106,-24.046,21.621,-43.804
C02454=1016.530,-67.505,-114.138,-24.046,21.621,-43.798
C02455=1016.533,-67.096,-114.170,-24.047,21.620,-43.791
C02456=1016.536,-66.686,-114.201,-24.048,21.620,-43.785
C02457=1016.539,-66.276,-114.233,-24.049,21.619,-43.780
C02458=1016.542,-65.867,-114.264,-24.049,21.618,-43.774
C02459=1016.544,-65.458,-114.295,-24.050,21.617,-43.768
C02460=1016.547,-65.050,-114.327,-24.051,21.617,-43.761
C02461=1016.550,-64.641,-114.358,-24.052,21.616,-43.756
C02462=1016.553,-64.234,-114.390,-24.053,21.615,-43.750
C02463=1016.556,-63.827,-114.421,-24.053,21.615,-43.744
C02464=1016.558,-63.420,-114.453,-24.054,21.615,-43.737
C02465=1016.562,-63.014,-114.483,-24.055,21.614,-43.732
C02466=1016.564,-62.608,-114.515,-24.056,21.613,-43.726
C02467=1016.567,-62.202,-114.546,-24.057,21.612,-43.720
C02468=1016.570,-61.798,-114.578,-24.057,21.611,-43.715
C02469=1016.573,-61.393,-114.609,-24.058,21.611,-43.708
C02470=1016.574,-60.990,-114.640,-24.059,21.610,-43.702
C02471=1016.578,-60.587,-114.671,-24.060,21.610,-43.697
C02472=1016.580,-60.185,-114.702,-24.061,21.610,-43.691
C02473=1016.582,-59.783,-114.734,-24.061,21.609,-43.686
C02474=1016.585,-59.382,-114.764,-24.062,21.608,-43.680
C02475=1016.588,-58.981,-114.796,-24.063,21.608,-43.673
C02476=1016.590,-58.581,-114.826,-24.064,21.607,-43.667
C02477=1016.593,-58.181,-114.858,-24.064,21.606,-43.662
C02478=1016.595,-57.781,-114.889,-24.065,21.606,-43.656
C02479=1016.597,-57.383,-114.920,-24.066,21.605,-43.651
C02480=1016.599,-56.985,-114.951,-24.067,21.604,-43.645
C02481=1016.601,-56.587,-114.982,-24.067,21.603,-43.639
C02482=1016.603,-56.189,-115.013,-24.068,21.603,-43.632
C02483=1016.606,-55.792,-115.044,-24.069,21.602,-43.627
C02484=1016.607,-55.394,-115.075,-24.070,21.603,-43.621
C02485=1016.610,-54.997,-115.106,-24.071,21.602,-43.616
C02486=1016.612,-54.600,-115.137,-24.071,21.601,-43.610
C02487=1016.615,-54.203,-115.168,-24.072,21.600,-43.604
C02488=1016.616,-53.806,-115.199,-24.073,21.599,-43.599
C02489=1016.619,-53.409,-115.231,-24.073,21.599,-43.593
C02490=1016.621,-53.012,-115.262,-24.074,21.598,-43.588
C02491=1016.623,-52.615,-115.292,-24.075,21.598,-43.581
C02492=1016.625,-52.218,-115.324,-24.076,21.598,-43.575
C02493=1016.627,-51.821,-115.355,-24.077,21.597,-43.570
C02494=1016.629,-51.425,-115.386,-24.077,21.596,-43.564
C02495=1016.631,-51.028,-115.417,-24.078,21.595,-43.558
C02496=1016.633,-50.631,-115.448,-24.079,21.595,-43.553
C02497=1016.635,-50.233,-115.479,-24.080,21.594,-43.547
C02498=1016.637,-49.836,-115.510,-24.080,21.593,-43.542
C02499=1016.638,-49.439,-115.542,-24.081,21.592,-43.536
C02500=1016.641,-49.043,-115.573,-24.082,21.592,-43.531
C02501=1016.642,-48.645,-115.604,-24.083,21.592,-43.525
C02502=1016.644,-48.248,-115.636,-24.084,21.592,-43.518
C02503=1016.645,-47.851,-115.667,-24.084,21.591,-43.512
C02504=1016.648,-47.454,-115.698,-24.085,21.590,-43.507
C02505=1016.649,-47.057,-115.730,-24.086,21.589,-43.501
C02506=1016.650,-46.660,-115.761,-24.086,21.588,-43.496
C02507=1016.653,-46.262,-115.793,-24.087,21.589,-43.490
C02508=1016.654,-45.865,-115.824,-24.088,21.588,-43.485
C02509=1016.656,-45.468,-115.855,-24.089,21.587,-43.479
C02510=1016.657,-45.071,-115.886,-24.089,21.586,-43.473
C02511=1016.660,-44.673,-115.918,-24.090,21.585,-43.468
C02512=1016.661,-44.276,-115.950,-24.091,21.585,-43.462
C02513=1016.663,-43.879,-115.981,-24.092,21.585,-43.457
C02514=1016.664,-43.482,-116.013,-24.092,21.584,-43.451
C02515=1016.665,-43.085,-116.044,-24.093,21.584,-43.444
C02516=1016.667,-42.687,-116.076,-24.094,21.583,-43.439
C02517=1016.668,-42.290,-116.108,-24.095,21.582,-43.433
C02518=1016.670,-41.893,-116.140,-24.096,21.582,-43.427
C02519=1016.671,-41.496,-116.171,-24.096,21.582,-43.422
C02520=1016.673,-41.098,-116.202,-24.097,21.581,-43.417
C02521=1016.675,-40.701,-116.234,-24.098,21.580,-43.411
C02522=1016.675,-40.304,-116.266,-24.099,21.579,-43.405
C02523=1016.677,-39.907,-116.298,-24.099,21.579,-43.400
C02524=1016.678,-39.510,-116.329,-24.100,21.578,-43.394
C02525=1016.679,-39.111,-116.361,-24.101,21.578,-43.389
C02526=1016.681,-38.714,-116.393,-24.102,21.577,-43.383
C02527=1016.682,-38.317,-116.425,-24.102,21.576,-43.378
C02528=1016.683,-37.920,-116.457,-24.103,21.576,-43.372
C02529=1016.685,-37.523,-116.488,-24.104,21.575,-43.366
C02530=1016.686,-37.125,-116.520,-24.105,21.575,-43.361
C02531=1016.687,-36.727,-116.552,-24.105,21.574,-43.356
C02532=1016.688,-36.330,-116.584,-24.106,21.573,-43.350
C02533=1016.689,-35.933,-116.616,-24.107,21.573,-43.344
C02534=1016.691,-35.536,-116.648,-24.107,21.572,-43.339
C02535=1016.692,-35.138,-116.680,-24.108,21.572,-43.334
C02536=1016.692,-34.741,-116.712,-24.109,21.571,-43.328
C02537=1016.694,-34.344,-116.743,-24.110,21.571,-43.321
C02538=1016.694,-33.946,-116.775,-24.111,21.570,-43.315
C02539=1016.696,-33.548,-116.808,-24.111,21.570,-43.310
C02540=1016.697,-33.151,-116.840,-24.112,21.570,-43.304
C02541=1016.698,-32.754,-116.872,-24.113,21.569,-43.299
C02542=1016.699,-32.357,-116.904,-24.114,21.568,-43.293
C02543=1016.700,-31.960,-116.936,-24.114,21.567,-43.287
C02544=1016.701,-31.561,-116.968,-24.115,21.568,-43.282
C02545=1016.701,-31.164,-117.000,-24.116,21.567,-43.277
C02546=1016.702,-30.767,-117.032,-24.117,21.566,-43.271
C02547=1016.703,-30.369,-117.064,-24.117,21.565,-43.265
C02548=1016.704,-29.972,-117.097,-24.118,21.565,-43.260
C02549=1016.705,-29.575,-117.129,-24.119,21.565,-43.255
C02550=1016.706,-29.177,-117.161,-24.120,21.564,-43.249
C02551=1016.707,-28.780,-117.194,-24.120,21.563,-43.243
C02552=1016.707,-28.383,-117.226,-24.121,21.562,-43.238
C02553=1016.708,-27.985,-117.258,-24.122,21.562,-43.232
C02554=1016.708,-27.588,-117.291,-24.123,21.562,-43.227
C02555=1016.709,-27.189,-117.322,-24.123,21.561,-43.221
C02556=1016.710,-26.792,-117.355,-24.124,21.560,-43.217
C02557=1016.711,-26.395,-117.387,-24.125,21.560,-43.212
C02558=1016.711,-25.997,-117.420,-24.125,21.559,-43.206
C02559=1016.712,-25.600,-117.452,-24.126,21.558,-43.201
C02560=1016.712,-25.203,-117.484,-24.127,21.558,-43.195
C02561=1016.713,-24.804,-117.517,-24.128,21.558,-43.190
C02562=1016.714,-24.407,-117.549,-24.128,21.557,-43.184
C02563=1016.715,-24.010,-117.582,-24.129,21.556,-43.178
C02564=1016.715,-23.612,-117.614,-24.130,21.556,-43.173
C02565=1016.715,-23.215,-117.646,-24.131,21.555,-43.168
C02566=1016.715,-22.818,-117.679,-24.131,21.555,-43.162
C02567=1016.716,-22.420,-117.711,-24.132,21.554,-43.156
C02568=1016.717,-22.022,-117.745,-24.133,21.554,-43.151
C02569=1016.717,-21.624,-117.777,-24.134,21.553,-43.146
C02570=1016.718,-21.227,-117.810,-24.134,21.552,-43.140
C02571=1016.718,-20.830,-117.842,-24.135,21.553,-43.135
C02572=1016.718,-20.432,-117.875,-24.136,21.552,-43.129
C02573=1016.718,-20.035,-117.907,-24.136,21.551,-43.123
C02574=1016.719,-19.623,-117.941,-24.138,21.551,-43.116
C02575=1016.719,-19.374,-117.962,-24.138,21.550,-43.113
C02576=1016.719,-19.087,-117.985,-24.139,21.550,-43.109
C02577=1016.720,-18.774,-118.011,-24.139,21.550,-43.107
C02578=1016.720,-18.463,-118.037,-24.139,21.549,-43.105
C02579=1016.720,-18.176,-118.061,-24.139,21.549,-43.101
C02580=1016.720,-17.928,-118.081,-24.140,21.548,-43.098
C02581=1016.720,-17.517,-118.115,-24.141,21.547,-43.090
C02582=1016.721,-17.119,-118.148,-24.142,21.548,-43.085
C02583=1016.721,-16.721,-118.181,-24.142,21.547,-43.079
C02584=1016.721,-16.322,-118.213,-24.143,21.546,-43.074
C02585=1016.721,-15.923,-118.246,-24.144,21.546,-43.068
C02586=1016.721,-15.523,-118.280,-24.145,21.545,-43.063
C02587=1016.722,-15.120,-118.313,-24.145,21.545,-43.057
C02588=1016.721,-14.714,-118.346,-24.146,21.544,-43.052
C02589=1016.721,-14.305,-118.380,-24.147,21.544,-43.046
C02590=1016.722,-13.894,-118.415,-24.148,21.543,-43.041
C02591=1016.721,-13.480,-118.449,-24.148,21.543,-43.035
C02592=1016.722,-13.062,-118.484,-24.149,21.542,-43.029
C02593=1016.722,-12.642,-118.518,-24.150,21.542,-43.024
C02594=1016.722,-12.432,-118.536,-24.150,21.541,-43.022
C02595=1016.722,-12.220,-118.553,-24.151,21.541,-43.019
C02596=1016.721,-12.008,-118.571,-24.151,21.540,-43.016
C02597=1016.722,-11.796,-118.589,-24.151,21.540,-43.013
C02598=1016.722,-11.583,-118.607,-24.152,21.540,-43.011
C02599=1016.722,-11.370,-118.624,-24.152,21.540,-43.007
C02600=1016.722,-11.156,-118.642,-24.152,21.539,-43.006
C02601=1016.722,-10.942,-118.660,-24.153,21.539,-43.002
C02602=1016.721,-10.727,-118.678,-24.153,21.539,-42.998
C02603=1016.722,-10.512,-118.696,-24.154,21.538,-42.996
C02604=1016.721,-10.297,-118.713,-24.154,21.539,-42.993
C02605=1016.721,-10.082,-118.732,-24.154,21.538,-42.991
C02606=1016.721,-9.866,-118.749,-24.155,21.538,-42.987
C02607=1016.721,-9.649,-118.767,-24.155,21.538,-42.985
C02608=1016.721,-9.434,-118.786,-24.156,21.537,-42.982
C02609=1016.721,-9.217,-118.804,-24.156,21.537,-42.980
C02610=1016.721,-9.000,-118.822,-24.156,21.536,-42.976
C02611=1016.721,-8.784,-118.839,-24.157,21.537,-42.973
C02612=1016.720,-8.567,-118.858,-24.157,21.536,-42.971
C02613=1016.721,-8.350,-118.876,-24.158,21.536,-42.967
C02614=1016.721,-8.134,-118.894,-24.158,21.536,-42.965
C02615=1016.720,-7.916,-118.912,-24.158,21.535,-42.961
C02616=1016.720,-7.698,-118.930,-24.159,21.535,-42.959
C02617=1016.720,-7.479,-118.949,-24.159,21.534,-42.956
C02618=1016.720,-7.259,-118.967,-24.160,21.535,-42.952
C02619=1016.720,-7.037,-118.985,-24.160,21.534,-42.950
C02620=1016.719,-6.815,-119.004,-24.160,21.534,-42.947
C02621=1016.719,-6.591,-119.023,-24.161,21.533,-42.944
C02622=1016.719,-6.368,-119.042,-24.161,21.533,-42.941
C02623=1016.719,-6.143,-119.061,-24.161,21.533,-42.939
C02624=1016.719,-5.919,-119.079,-24.162,21.533,-42.935
C02625=1016.718,-5.695,-119.098,-24.162,21.532,-42.934
C02626=1016.718,-5.471,-119.117,-24.163,21.532,-42.930
C02627=1016.718,-5.249,-119.136,-24.163,21.532,-42.927
C02628=1016.719,-5.027,-119.154,-24.163,21.532,-42.925
C02629=1016.718,-4.807,-119.173,-24.164,21.531,-42.921
C02630=1016.718,-4.589,-119.191,-24.164,21.531,-42.919
C02631=1016.718,-4.372,-119.209,-24.165,21.531,-42.915
C02632=1016.717,-4.157,-119.227,-24.165,21.530,-42.913
C02633=1016.717,-3.943,-119.246,-24.165,21.530,-42.910
C02634=1016.717,-3.731,-119.263,-24.166,21.530,-42.908
C02635=1016.716,-3.520,-119.281,-24.166,21.530,-42.904
C02636=1016.717,-3.098,-119.316,-24.167,21.529,-42.899
C02637=1016.716,-2.679,-119.352,-24.168,21.529,-42.893
C02638=1016.715,-2.262,-119.386,-24.169,21.529,-42.888
C02639=1016.715,-1.847,-119.422,-24.169,21.528,-42.882
C02640=1016.713,-1.434,-119.456,-24.170,21.527,-42.877
C02641=1016.714,-1.024,-119.491,-24.171,21.527,-42.872
C02642=1016.713,-0.616,-119.525,-24.171,21.526,-42.867
C02643=1016.712,-0.211,-119.560,-24.172,21.525,-42.862
C02644=1016.711,0.193,-119.594,-24.173,21.525,-42.857
C02645=1016.711,0.594,-119.627,-24.173,21.525,-42.851
C02646=1016.711,0.994,-119.661,-24.174,21.525,-42.846
C02647=1016.710,1.393,-119.695,-24.175,21.523,-42.841
C02648=1016.709,1.791,-119.729,-24.175,21.524,-42.836
C02649=1016.709,2.177,-119.761,-24.176,21.523,-42.833
C02650=1016.708,2.530,-119.792,-24.177,21.522,-42.827
C02651=1016.708,2.853,-119.819,-24.177,21.522,-42.823
C02652=1016.707,3.166,-119.846,-24.178,21.521,-42.817
C02653=1016.707,3.494,-119.873,-24.179,21.521,-42.812
C02654=1016.706,3.853,-119.904,-24.179,21.521,-42.809
C02655=1016.705,4.242,-119.936,-24.180,21.520,-42.805
C02656=1016.704,4.638,-119.971,-24.180,21.519,-42.799
C02657=1016.703,5.034,-120.004,-24.181,21.520,-42.794
C02658=1016.702,5.429,-120.037,-24.182,21.519,-42.790
C02659=1016.702,5.823,-120.072,-24.182,21.518,-42.785
C02660=1016.701,6.217,-120.105,-24.183,21.519,-42.779
C02661=1016.699,6.610,-120.138,-24.184,21.517,-42.775
C02662=1016.699,7.002,-120.172,-24.185,21.517,-42.770
C02663=1016.698,7.393,-120.205,-24.185,21.517,-42.764
C02664=1016.698,7.781,-120.238,-24.186,21.516,-42.761
C02665=1016.696,8.164,-120.271,-24.187,21.516,-42.755
C02666=1016.696,8.545,-120.304,-24.187,21.515,-42.751
C02667=1016.695,8.923,-120.335,-24.188,21.515,-42.746
C02668=1016.694,9.299,-120.368,-24.189,21.514,-42.740
C02669=1016.693,9.675,-120.400,-24.189,21.514,-42.737
C02670=1016.692,10.052,-120.432,-24.190,21.513,-42.731
C02671=1016.691,10.430,-120.465,-24.191,21.513,-42.726
C02672=1016.690,10.811,-120.497,-24.191,21.513,-42.722
C02673=1016.689,11.194,-120.530,-24.192,21.512,-42.716
C02674=1016.687,11.580,-120.563,-24.192,21.511,-42.713
C02675=1016.686,11.966,-120.596,-24.193,21.512,-42.707
C02676=1016.685,12.352,-120.630,-24.193,21.510,-42.703
C02677=1016.684,12.738,-120.662,-24.194,21.510,-42.698
C02678=1016.683,13.125,-120.696,-24.195,21.511,-42.693
C02679=1016.682,13.513,-120.729,-24.196,21.509,-42.689
C02680=1016.680,13.899,-120.763,-24.196,21.509,-42.683
C02681=1016.680,14.288,-120.796,-24.197,21.509,-42.680
C02682=1016.679,14.676,-120.829,-24.198,21.508,-42.674
C02683=1016.677,15.064,-120.863,-24.198,21.508,-42.670
C02684=1016.677,15.454,-120.896,-24.199,21.507,-42.665
C02685=1016.675,15.844,-120.930,-24.200,21.507,-42.659
C02686=1016.674,16.235,-120.964,-24.200,21.506,-42.656
C02687=1016.672,16.627,-120.997,-24.201,21.506,-42.650
C02688=1016.671,17.019,-121.031,-24.201,21.505,-42.646
C02689=1016.670,17.413,-121.065,-24.202,21.505,-42.641
C02690=1016.668,17.807,-121.099,-24.203,21.505,-42.635
C02691=1016.667,18.202,-121.133,-24.203,21.504,-42.632
C02692=1016.666,18.598,-121.168,-24.204,21.503,-42.626
C02693=1016.664,18.994,-121.202,-24.205,21.503,-42.622
C02694=1016.663,19.392,-121.236,-24.205,21.503,-42.617
C02695=1016.662,19.602,-121.255,-24.206,21.503,-42.613
C02696=1016.662,19.839,-121.275,-24.206,21.502,-42.610
C02697=1016.660,20.104,-121.298,-24.207,21.503,-42.606
C02698=1016.659,20.392,-121.322,-24.207,21.501,-42.604
C02699=1016.657,20.688,-121.348,-24.207,21.501,-42.602
C02700=1016.657,20.980,-121.374,-24.208,21.502,-42.599
C02701=1016.656,21.252,-121.397,-24.208,21.501,-42.597
C02702=1016.654,21.496,-121.418,-24.209,21.501,-42.593
C02703=1016.653,21.910,-121.455,-24.210,21.501,-42.586
C02704=1016.652,22.285,-121.487,-24.210,21.500,-42.584
C02705=1016.651,22.607,-121.515,-24.211,21.500,-42.580
C02706=1016.649,22.874,-121.538,-24.211,21.500,-42.577
C02707=1016.648,23.105,-121.559,-24.211,21.499,-42.573
C02708=1016.648,23.340,-121.579,-24.212,21.498,-42.567
C02709=1016.646,23.611,-121.602,-24.213,21.498,-42.564
C02710=1016.646,23.942,-121.631,-24.213,21.498,-42.562
C02711=1016.644,24.325,-121.664,-24.213,21.497,-42.558
C02712=1016.642,24.724,-121.699,-24.214,21.497,-42.553
C02713=1016.641,25.123,-121.734,-24.215,21.497,-42.549
C02714=1016.638,25.523,-121.770,-24.215,21.496,-42.543
C02715=1016.637,25.923,-121.804,-24.216,21.496,-42.540
C02716=1016.635,26.322,-121.839,-24.217,21.496,-42.534
C02717=1016.633,26.720,-121.873,-24.218,21.495,-42.529
C02718=1016.631,27.119,-121.908,-24.218,21.494,-42.525
C02719=1016.630,27.519,-121.943,-24.219,21.495,-42.520
C02720=1016.628,27.919,-121.977,-24.219,21.493,-42.516
C02721=1016.626,28.319,-122.013,-24.220,21.493,-42.510
C02722=1016.624,28.718,-122.048,-24.221,21.493,-42.507
C02723=1016.623,29.117,-122.083,-24.221,21.492,-42.501
C02724=1016.620,29.517,-122.118,-24.222,21.492,-42.497
C02725=1016.619,29.917,-122.153,-24.223,21.492,-42.492
C02726=1016.617,30.316,-122.188,-24.223,21.491,-42.488
C02727=1016.615,30.715,-122.223,-24.224,21.491,-42.483
C02728=1016.613,31.115,-122.258,-24.224,21.490,-42.479
C02729=1016.610,31.515,-122.293,-24.225,21.490,-42.474
C02730=1016.609,31.914,-122.328,-24.226,21.489,-42.469
C02731=1016.607,32.313,-122.364,-24.226,21.489,-42.464
C02732=1016.605,32.713,-122.398,-24.227,21.489,-42.461
C02733=1016.603,33.114,-122.434,-24.228,21.489,-42.455
C02734=1016.601,33.513,-122.469,-24.228,21.487,-42.451
C02735=1016.599,33.912,-122.504,-24.229,21.488,-42.446
C02736=1016.596,34.312,-122.539,-24.229,21.487,-42.442
C02737=1016.595,34.712,-122.574,-24.230,21.486,-42.437
C02738=1016.592,35.111,-122.609,-24.231,21.486,-42.433
C02739=1016.590,35.511,-122.645,-24.231,21.486,-42.428
C02740=1016.588,35.912,-122.680,-24.232,21.486,-42.424
C02741=1016.586,36.311,-122.716,-24.233,21.485,-42.418
C02742=1016.584,36.710,-122.751,-24.233,21.484,-42.414
C02743=1016.582,37.111,-122.785,-24.234,21.485,-42.409
C02744=1016.579,37.510,-122.821,-24.235,21.484,-42.405
C02745=1016.578,37.910,-122.857,-24.235,21.483,-42.400
C02746=1016.575,38.310,-122.892,-24.236,21.483,-42.396
C02747=1016.573,38.710,-122.927,-24.237,21.483,-42.391
C02748=1016.570,39.110,-122.963,-24.237,21.483,-42.387
C02749=1016.568,39.510,-122.997,-24.238,21.482,-42.383
C02750=1016.566,39.910,-123.033,-24.238,21.481,-42.378
C02751=1016.564,40.309,-123.069,-24.239,21.481,-42.374
C02752=1016.561,40.710,-123.104,-24.240,21.481,-42.369
C02753=1016.559,41.109,-123.139,-24.240,21.481,-42.365
C02754=1016.557,41.509,-123.175,-24.241,21.480,-42.359
C02755=1016.554,41.909,-123.211,-24.241,21.479,-42.356
C02756=1016.551,42.309,-123.246,-24.242,21.479,-42.352
C02757=1016.549,42.709,-123.282,-24.243,21.479,-42.347
C02758=1016.547,43.109,-123.317,-24.243,21.479,-42.343
C02759=1016.544,43.510,-123.353,-24.244,21.479,-42.338
C02760=1016.541,43.909,-123.388,-24.244,21.477,-42.333
C02761=1016.539,44.309,-123.424,-24.245,21.477,-42.330
C02762=1016.536,44.710,-123.460,-24.246,21.477,-42.325
C02763=1016.534,45.109,-123.495,-24.246,21.477,-42.321
C02764=1016.532,45.509,-123.531,-24.247,21.477,-42.316
C02765=1016.529,45.910,-123.566,-24.247,21.475,-42.311
C02766=1016.527,46.310,-123.602,-24.248,21.475,-42.308
C02767=1016.524,46.710,-123.638,-24.249,21.475,-42.302
C02768=1016.521,47.110,-123.673,-24.249,21.475,-42.299
C02769=1016.518,47.510,-123.709,-24.250,21.474,-42.295
C02770=1016.516,47.910,-123.745,-24.251,21.474,-42.290
C02771=1016.513,48.310,-123.780,-24.251,21.474,-42.286
C02772=1016.510,48.710,-123.816,-24.251,21.472,-42.282
C02773=1016.508,49.110,-123.852,-24.252,21.473,-42.277
C02774=1016.505,49.511,-123.888,-24.253,21.472,-42.273
C02775=1016.502,49.910,-123.923,-24.254,21.472,-42.268
C02776=1016.499,50.310,-123.959,-24.254,21.472,-42.264
C02777=1016.496,50.711,-123.995,-24.255,21.471,-42.260
C02778=1016.494,51.111,-124.031,-24.255,21.471,-42.255
C02779=1016.491,51.511,-124.067,-24.256,21.471,-42.251
C02780=1016.488,51.911,-124.102,-24.256,21.470,-42.247
C02781=1016.485,52.312,-124.139,-24.257,21.469,-42.243
C02782=1016.482,52.712,-124.175,-24.258,21.469,-42.238
C02783=1016.479,53.112,-124.210,-24.258,21.469,-42.234
C02784=1016.476,53.512,-124.246,-24.259,21.468,-42.230
C02785=1016.474,53.912,-124.282,-24.259,21.468,-42.225
C02786=1016.471,54.312,-124.318,-24.260,21.468,-42.221
C02787=1016.467,54.713,-124.354,-24.260,21.468,-42.218
C02788=1016.464,55.112,-124.390,-24.261,21.468,-42.212
C02789=1016.462,55.513,-124.426,-24.262,21.467,-42.209
C02790=1016.459,55.913,-124.462,-24.262,21.467,-42.205
C02791=1016.456,56.313,-124.498,-24.263,21.465,-42.201
C02792=1016.452,56.713,-124.534,-24.264,21.466,-42.196
C02793=1016.449,57.113,-124.570,-24.264,21.465,-42.192
C02794=1016.447,57.514,-124.606,-24.264,21.465,-42.188
C02795=1016.444,57.914,-124.642,-24.265,21.465,-42.183
C02796=1016.440,58.314,-124.678,-24.266,21.464,-42.179
C02797=1016.437,58.714,-124.714,-24.266,21.464,-42.175
C02798=1016.434,59.114,-124.750,-24.267,21.463,-42.172
C02799=1016.430,59.514,-124.786,-24.268,21.464,-42.166
C02800=1016.428,59.915,-124.823,-24.268,21.463,-42.163
C02801=1016.424,60.315,-124.858,-24.269,21.463,-42.159
C02802=1016.421,60.715,-124.894,-24.269,21.462,-42.155
C02803=1016.418,61.115,-124.931,-24.270,21.462,-42.150
C02804=1016.414,61.515,-124.967,-24.270,21.462,-42.146
C02805=1016.411,61.915,-125.003,-24.271,21.461,-42.142
C02806=1016.408,62.316,-125.039,-24.271,21.461,-42.139
C02807=1016.405,62.735,-125.077,-24.272,21.460,-42.133
C02808=1016.402,62.988,-125.100,-24.272,21.460,-42.131
C02809=1016.400,63.256,-125.125,-24.273,21.460,-42.129
C02810=1016.398,63.506,-125.147,-24.273,21.459,-42.127
C02811=1016.397,63.723,-125.167,-24.274,21.460,-42.124
C02812=1016.395,63.930,-125.186,-24.274,21.460,-42.122
C02813=1016.392,64.148,-125.205,-24.274,21.459,-42.120
C02814=1016.391,64.377,-125.226,-24.274,21.459,-42.116
C02815=1016.389,64.613,-125.248,-24.275,21.459,-42.115
C02816=1016.387,64.849,-125.268,-24.275,21.458,-42.113
C02817=1016.385,65.079,-125.289,-24.275,21.458,-42.111
C02818=1016.383,65.301,-125.310,-24.276,21.459,-42.108
C02819=1016.381,65.513,-125.329,-24.276,21.458,-42.106
C02820=1016.377,65.921,-125.366,-24.277,21.458,-42.102
C02821=1016.375,66.320,-125.402,-24.277,21.457,-42.098
C02822=1016.371,66.720,-125.439,-24.278,21.457,-42.094
C02823=1016.368,67.123,-125.475,-24.278,21.457,-42.089
C02824=1016.364,67.526,-125.511,-24.279,21.457,-42.085
C02825=1016.360,67.930,-125.548,-24.279,21.456,-42.082
C02826=1016.357,68.336,-125.585,-24.280,21.456,-42.078
C02827=1016.353,68.743,-125.622,-24.280,21.455,-42.074
C02828=1016.349,69.152,-125.659,-24.281,21.455,-42.069
C02829=1016.345,69.563,-125.697,-24.282,21.455,-42.065
C02830=1016.342,69.974,-125.735,-24.282,21.454,-42.061
C02831=1016.338,70.385,-125.771,-24.283,21.454,-42.058
C02832=1016.334,70.796,-125.809,-24.283,21.453,-42.054
C02833=1016.331,71.207,-125.846,-24.284,21.454,-42.049
C02834=1016.326,71.618,-125.884,-24.285,21.453,-42.045
C02835=1016.323,72.030,-125.921,-24.285,21.453,-42.041
C02836=1016.319,72.444,-125.959,-24.285,21.452,-42.037
C02837=1016.315,72.859,-125.997,-24.286,21.452,-42.034
C02838=1016.311,73.277,-126.035,-24.287,21.452,-42.028
C02839=1016.307,73.698,-126.073,-24.287,21.452,-42.025
C02840=1016.305,73.908,-126.093,-24.288,21.451,-42.023
C02841=1016.303,74.121,-126.112,-24.288,21.451,-42.021
C02842=1016.301,74.333,-126.132,-24.288,21.451,-42.019
C02843=1016.299,74.546,-126.151,-24.288,21.451,-42.017
C02844=1016.297,74.759,-126.170,-24.289,21.450,-42.015
C02845=1016.295,74.974,-126.190,-24.289,21.451,-42.012
C02846=1016.292,75.186,-126.210,-24.289,21.451,-42.010
C02847=1016.290,75.399,-126.229,-24.290,21.450,-42.008
C02848=1016.287,75.819,-126.267,-24.290,21.450,-42.004
C02849=1016.283,76.230,-126.305,-24.291,21.449,-42.001
C02850=1016.279,76.633,-126.341,-24.291,21.449,-41.997
C02851=1016.275,77.027,-126.377,-24.292,21.449,-41.994
C02852=1016.270,77.416,-126.413,-24.292,21.448,-41.989
C02853=1016.268,77.802,-126.448,-24.293,21.447,-41.986
C02854=1016.264,78.189,-126.484,-24.293,21.448,-41.980
C02855=1016.259,78.578,-126.520,-24.294,21.447,-41.977
C02856=1016.255,78.976,-126.556,-24.294,21.447,-41.973
C02857=1016.251,79.382,-126.593,-24.295,21.447,-41.970
C02858=1016.247,79.796,-126.631,-24.296,21.447,-41.966
C02859=1016.244,80.006,-126.650,-24.296,21.446,-41.964
C02860=1016.243,80.218,-126.670,-24.296,21.446,-41.962
C02861=1016.240,80.431,-126.689,-24.296,21.446,-41.960
C02862=1016.238,80.643,-126.709,-24.297,21.446,-41.958
C02863=1016.236,80.856,-126.728,-24.297,21.445,-41.956
C02864=1016.234,81.069,-126.748,-24.297,21.445,-41.955
C02865=1016.232,81.281,-126.768,-24.297,21.445,-41.953
C02866=1016.230,81.493,-126.787,-24.298,21.445,-41.951
C02867=1016.228,81.706,-126.806,-24.298,21.445,-41.949
C02868=1016.225,81.917,-126.825,-24.298,21.444,-41.947
C02869=1016.223,82.128,-126.845,-24.299,21.445,-41.944
C02870=1016.221,82.341,-126.864,-24.299,21.444,-41.942
C02871=1016.216,82.761,-126.903,-24.299,21.444,-41.938
C02872=1016.212,83.182,-126.942,-24.300,21.444,-41.935
C02873=1016.207,83.601,-126.980,-24.300,21.444,-41.931
C02874=1016.202,84.017,-127.019,-24.301,21.443,-41.927
C02875=1016.199,84.433,-127.057,-24.301,21.443,-41.923
C02876=1016.194,84.848,-127.095,-24.302,21.443,-41.920
C02877=1016.190,85.260,-127.133,-24.302,21.442,-41.916
C02878=1016.185,85.670,-127.171,-24.303,21.442,-41.912
C02879=1016.180,86.080,-127.208,-24.303,21.441,-41.908
C02880=1016.176,86.487,-127.245,-24.304,21.442,-41.905
C02881=1016.171,86.893,-127.283,-24.304,21.441,-41.901
C02882=1016.167,87.296,-127.320,-24.305,21.441,-41.898
C02883=1016.163,87.692,-127.357,-24.305,21.440,-41.894
C02884=1016.158,88.080,-127.392,-24.306,21.440,-41.890
C02885=1016.154,88.463,-127.428,-24.307,21.440,-41.887
C02886=1016.149,88.846,-127.463,-24.307,21.440,-41.883
C02887=1016.146,89.233,-127.499,-24.308,21.439,-41.879
C02888=1016.141,89.625,-127.535,-24.308,21.439,-41.875
C02889=1016.136,90.023,-127.571,-24.309,21.439,-41.872
C02890=1016.132,90.422,-127.609,-24.309,21.439,-41.868
C02891=1016.128,90.822,-127.645,-24.310,21.438,-41.865
C02892=1016.123,91.222,-127.682,-24.310,21.438,-41.861
C02893=1016.118,91.620,-127.719,-24.311,21.438,-41.857
C02894=1016.114,92.019,-127.756,-24.311,21.438,-41.854
C02895=1016.109,92.418,-127.793,-24.312,21.437,-41.850
C02896=1016.105,92.817,-127.830,-24.312,21.437,-41.846
C02897=1016.099,93.217,-127.867,-24.312,21.437,-41.844
C02898=1016.095,93.616,-127.904,-24.313,21.436,-41.841
C02899=1016.090,94.014,-127.940,-24.313,21.436,-41.837
C02900=1016.085,94.414,-127.977,-24.314,21.435,-41.833
C02901=1016.081,94.812,-128.014,-24.315,21.436,-41.830
C02902=1016.076,95.211,-128.051,-24.315,21.435,-41.826
C02903=1016.072,95.610,-128.088,-24.316,21.435,-41.822
C02904=1016.066,96.009,-128.125,-24.316,21.435,-41.819
C02905=1016.062,96.408,-128.162,-24.317,21.435,-41.815
C02906=1016.056,96.807,-128.199,-24.317,21.434,-41.811
C02907=1016.052,97.206,-128.235,-24.318,21.434,-41.808
C02908=1016.046,97.604,-128.272,-24.318,21.433,-41.806
C02909=1016.042,98.003,-128.310,-24.318,21.433,-41.802
C02910=1016.037,98.402,-128.346,-24.319,21.432,-41.798
C02911=1016.032,98.801,-128.383,-24.319,21.433,-41.795
C02912=1016.027,99.200,-128.420,-24.320,21.432,-41.791
C02913=1016.023,99.599,-128.457,-24.320,21.432,-41.787
C02914=1016.017,99.997,-128.494,-24.321,21.432,-41.784
C02915=1016.012,100.396,-128.531,-24.322,21.432,-41.780
C02916=1016.007,100.795,-128.568,-24.322,21.431,-41.778
C02917=1016.002,101.194,-128.605,-24.322,21.431,-41.775
C02918=1015.997,101.592,-128.642,-24.323,21.431,-41.771
C02919=1015.992,101.991,-128.679,-24.323,21.430,-41.767
C02920=1015.987,102.390,-128.716,-24.324,21.430,-41.763
C02921=1015.981,102.788,-128.753,-24.324,21.430,-41.760
C02922=1015.977,103.187,-128.790,-24.325,21.430,-41.756
C02923=1015.972,103.586,-128.828,-24.325,21.430,-41.754
C02924=1015.966,103.985,-128.864,-24.326,21.429,-41.751
C02925=1015.961,104.383,-128.901,-24.326,21.429,-41.747
C02926=1015.956,104.781,-128.938,-24.327,21.429,-41.743
C02927=1015.950,105.180,-128.975,-24.327,21.429,-41.740
C02928=1015.945,105.579,-129.012,-24.328,21.428,-41.736
C02929=1015.940,105.978,-129.050,-24.328,21.428,-41.734
C02930=1015.935,106.376,-129.086,-24.328,21.427,-41.730
C02931=1015.930,106.774,-129.124,-24.329,21.427,-41.727
C02932=1015.924,107.173,-129.161,-24.330,21.427,-41.723
C02933=1015.918,107.572,-129.198,-24.330,21.427,-41.719
C02934=1015.913,107.970,-129.235,-24.330,21.426,-41.717
C02935=1015.908,108.369,-129.272,-24.331,21.426,-41.714
C02936=1015.902,108.767,-129.309,-24.331,21.426,-41.710
C02937=1015.897,109.166,-129.347,-24.332,21.426,-41.707
C02938=1015.891,109.565,-129.383,-24.332,21.426,-41.703
C02939=1015.886,109.963,-129.421,-24.333,21.425,-41.701
C02940=1015.880,110.362,-129.458,-24.333,21.425,-41.697
C02941=1015.875,110.760,-129.495,-24.334,21.425,-41.694
C02942=1015.869,111.158,-129.533,-24.334,21.425,-41.690
C02943=1015.864,111.557,-129.569,-24.334,21.424,-41.688
C02944=1015.858,111.956,-129.606,-24.335,21.423,-41.684
C02945=1015.852,112.354,-129.643,-24.335,21.424,-41.681
C02946=1015.847,112.752,-129.681,-24.336,21.423,-41.677
C02947=1015.841,113.150,-129.718,-24.336,21.423,-41.675
C02948=1015.835,113.550,-129.754,-24.337,21.423,-41.671
C02949=1015.830,113.948,-129.792,-24.337,21.422,-41.668
C02950=1015.825,114.346,-129.829,-24.338,21.423,-41.664
C02951=1015.819,114.744,-129.866,-24.338,21.422,-41.662
C02952=1015.812,115.143,-129.904,-24.339,21.422,-41.659
C02953=1015.807,115.542,-129.940,-24.339,21.422,-41.655
C02954=1015.801,115.940,-129.978,-24.340,21.422,-41.652
C02955=1015.796,116.339,-130.015,-24.340,21.421,-41.649
C02956=1015.789,116.737,-130.053,-24.340,21.420,-41.646
C02957=1015.784,117.135,-130.090,-24.341,21.421,-41.642
C02958=1015.778,117.534,-130.126,-24.341,21.420,-41.638
C02959=1015.772,117.933,-130.164,-24.342,21.420,-41.637
C02960=1015.766,118.331,-130.201,-24.342,21.420,-41.633
C02961=1015.760,118.729,-130.238,-24.343,21.420,-41.629
C02962=1015.755,119.128,-130.276,-24.343,21.420,-41.626
C02963=1015.748,119.526,-130.313,-24.343,21.419,-41.624
C02964=1015.742,119.925,-130.350,-24.344,21.419,-41.620
C02965=1015.736,120.323,-130.388,-24.345,21.419,-41.617
C02966=1015.730,120.721,-130.425,-24.345,21.418,-41.614
C02967=1015.725,121.120,-130.462,-24.345,21.418,-41.611
C02968=1015.718,121.518,-130.500,-24.346,21.418,-41.607
C02969=1015.713,121.917,-130.537,-24.346,21.417,-41.605
C02970=1015.708,122.315,-130.574,-24.347,21.418,-41.602
C02971=1015.701,122.714,-130.612,-24.347,21.417,-41.598
C02972=1015.696,123.112,-130.650,-24.348,21.418,-41.595
C02973=1015.690,123.511,-130.687,-24.348,21.416,-41.592
C02974=1015.684,123.910,-130.725,-24.348,21.417,-41.589
C02975=1015.679,124.307,-130.763,-24.349,21.416,-41.585
C02976=1015.673,124.706,-130.801,-24.349,21.416,-41.583
C02977=1015.668,125.104,-130.838,-24.350,21.416,-41.580
C02978=1015.661,125.503,-130.876,-24.350,21.416,-41.576
C02979=1015.656,125.902,-130.913,-24.350,21.415,-41.574
C02980=1015.650,126.300,-130.951,-24.351,21.415,-41.571
C02981=1015.644,126.699,-130.988,-24.351,21.415,-41.567
C02982=1015.638,127.098,-131.026,-24.352,21.415,-41.565
C02983=1015.631,127.496,-131.064,-24.352,21.414,-41.561
C02984=1015.626,127.894,-131.101,-24.353,21.415,-41.558
C02985=1015.620,128.293,-131.139,-24.353,21.414,-41.555
C02986=1015.614,128.692,-131.177,-24.354,21.414,-41.552
C02987=1015.608,129.090,-131.214,-24.354,21.413,-41.550
C02988=1015.602,129.489,-131.252,-24.354,21.413,-41.547
C02989=1015.596,129.887,-131.290,-24.355,21.413,-41.543
C02990=1015.590,130.285,-131.327,-24.355,21.413,-41.541
C02991=1015.584,130.684,-131.365,-24.356,21.413,-41.538
C02992=1015.577,131.083,-131.402,-24.356,21.413,-41.534
C02993=1015.571,131.482,-131.440,-24.356,21.412,-41.532
C02994=1015.565,131.881,-131.478,-24.357,21.412,-41.528
C02995=1015.559,132.278,-131.515,-24.357,21.412,-41.525
C02996=1015.553,132.677,-131.552,-24.358,21.411,-41.523
C02997=1015.546,133.076,-131.590,-24.358,21.412,-41.519
C02998=1015.540,133.475,-131.628,-24.358,21.411,-41.517
C02999=1015.534,133.873,-131.666,-24.359,21.411,-41.514
C03000=1015.527,134.271,-131.704,-24.359,21.411,-41.510
C03001=1015.521,134.670,-131.742,-24.360,21.410,-41.508
C03002=1015.515,135.070,-131.779,-24.360,21.411,-41.505
C03003=1015.508,135.465,-131.816,-24.360,21.410,-41.502
C03004=1015.503,135.836,-131.851,-24.361,21.409,-41.500
C03005=1015.498,136.175,-131.883,-24.361,21.410,-41.497
C03006=1015.492,136.493,-131.913,-24.361,21.409,-41.495
C03007=1015.487,136.809,-131.944,-24.362,21.409,-41.491
C03008=1015.482,137.146,-131.976,-24.363,21.410,-41.488
C03009=1015.475,137.515,-132.010,-24.363,21.408,-41.486
C03010=1015.469,137.917,-132.048,-24.363,21.408,-41.484
C03011=1015.465,138.122,-132.067,-24.363,21.408,-41.482
C03012=1015.462,138.339,-132.089,-24.364,21.408,-41.480
C03013=1015.458,138.577,-132.111,-24.364,21.408,-41.478
C03014=1015.453,138.836,-132.136,-24.364,21.407,-41.476
C03015=1015.449,139.114,-132.162,-24.364,21.408,-41.475
C03016=1015.444,139.402,-132.189,-24.365,21.408,-41.473
C03017=1015.440,139.690,-132.216,-24.365,21.408,-41.471
C03018=1015.435,139.967,-132.242,-24.365,21.408,-41.470
C03019=1015.431,140.225,-132.266,-24.366,21.408,-41.468
C03020=1015.427,140.461,-132.289,-24.366,21.408,-41.466
C03021=1015.420,140.878,-132.328,-24.366,21.407,-41.462
C03022=1015.413,141.283,-132.367,-24.366,21.406,-41.460
C03023=1015.406,141.688,-132.405,-24.367,21.407,-41.457
C03024=1015.399,142.094,-132.443,-24.368,21.406,-41.453
C03025=1015.393,142.501,-132.482,-24.368,21.406,-41.451
C03026=1015.385,142.909,-132.521,-24.368,21.406,-41.448
C03027=1015.379,143.317,-132.559,-24.369,21.405,-41.445
C03028=1015.372,143.727,-132.599,-24.369,21.406,-41.442
C03029=1015.364,144.138,-132.637,-24.370,21.405,-41.438
C03030=1015.357,144.548,-132.676,-24.370,21.405,-41.436
C03031=1015.350,144.960,-132.715,-24.370,21.405,-41.432
C03032=1015.343,145.371,-132.754,-24.371,21.404,-41.431
C03033=1015.336,145.784,-132.794,-24.371,21.405,-41.427
C03034=1015.329,146.197,-132.832,-24.372,21.404,-41.424
C03035=1015.321,146.610,-132.872,-24.372,21.404,-41.422
C03036=1015.314,147.024,-132.910,-24.372,21.404,-41.418
C03037=1015.307,147.437,-132.949,-24.373,21.403,-41.416
C03038=1015.300,147.850,-132.989,-24.373,21.403,-41.412
C03039=1015.292,148.264,-133.028,-24.374,21.403,-41.409
C03040=1015.285,148.678,-133.067,-24.374,21.403,-41.407
C03041=1015.277,149.092,-133.107,-24.375,21.403,-41.403
C03042=1015.270,149.506,-133.146,-24.375,21.402,-41.401
C03043=1015.263,149.921,-133.185,-24.375,21.402,-41.398
C03044=1015.255,150.334,-133.224,-24.376,21.402,-41.394
C03045=1015.247,150.748,-133.263,-24.376,21.401,-41.392
C03046=1015.240,151.161,-133.302,-24.377,21.402,-41.389
C03047=1015.232,151.574,-133.342,-24.377,21.402,-41.387
C03048=1015.225,151.988,-133.381,-24.377,21.401,-41.383
C03049=1015.218,152.400,-133.420,-24.378,21.401,-41.381
C03050=1015.210,152.812,-133.459,-24.378,21.400,-41.377
C03051=1015.202,153.224,-133.498,-24.378,21.400,-41.375
C03052=1015.194,153.635,-133.537,-24.379,21.401,-41.372
C03053=1015.187,154.046,-133.576,-24.380,21.400,-41.368
C03054=1015.179,154.455,-133.615,-24.380,21.400,-41.366
C03055=1015.171,154.865,-133.653,-24.380,21.400,-41.363
C03056=1015.163,155.273,-133.693,-24.381,21.399,-41.361
C03057=1015.156,155.681,-133.731,-24.381,21.400,-41.358
C03058=1015.148,156.087,-133.769,-24.381,21.399,-41.355
C03059=1015.140,156.493,-133.808,-24.382,21.399,-41.352
C03060=1015.133,156.898,-133.846,-24.382,21.399,-41.350
C03061=1015.125,157.302,-133.884,-24.383,21.398,-41.346
C03062=1015.117,157.705,-133.923,-24.383,21.398,-41.344
C03063=1015.109,158.108,-133.961,-24.383,21.399,-41.341
C03064=1015.102,158.510,-133.999,-24.384,21.397,-41.339
C03065=1015.094,158.911,-134.037,-24.384,21.398,-41.335
C03066=1015.086,159.312,-134.075,-24.384,21.398,-41.333
C03067=1015.079,159.712,-134.113,-24.385,21.397,-41.330
C03068=1015.076,160.109,-134.154,-24.385,21.397,-41.328
C03069=1015.075,160.513,-134.197,-24.386,21.397,-41.325
C03070=1015.074,160.727,-134.218,-24.386,21.397,-41.324
C03071=1015.073,160.951,-134.242,-24.386,21.396,-41.322
C03072=1015.072,161.188,-134.267,-24.386,21.396,-41.320
C03073=1015.071,161.439,-134.294,-24.387,21.397,-41.319
C03074=1015.069,161.702,-134.320,-24.387,21.397,-41.317
C03075=1015.069,161.972,-134.349,-24.387,21.396,-41.315
C03076=1015.068,162.243,-134.378,-24.387,21.396,-41.313
C03077=1015.067,162.512,-134.405,-24.388,21.396,-41.311
C03078=1015.066,162.774,-134.432,-24.388,21.396,-41.309
C03079=1015.065,163.028,-134.460,-24.388,21.395,-41.308
C03080=1015.063,163.264,-134.484,-24.388,21.396,-41.306
C03081=1015.062,163.676,-134.527,-24.389,21.395,-41.304
C03082=1015.061,163.866,-134.547,-24.389,21.395,-41.302
C03083=1015.060,164.252,-134.587,-24.389,21.395,-41.300
C03084=1015.059,164.651,-134.629,-24.390,21.395,-41.297
C03085=1015.057,165.053,-134.672,-24.390,21.395,-41.295
C03086=1015.056,165.452,-134.714,-24.390,21.394,-41.291
C03087=1015.054,165.853,-134.756,-24.391,21.394,-41.289
C03088=1015.053,166.253,-134.798,-24.391,21.395,-41.286
C03089=1015.051,166.654,-134.840,-24.391,21.393,-41.284
C03090=1015.049,167.054,-134.882,-24.392,21.394,-41.280
C03091=1015.048,167.454,-134.924,-24.392,21.394,-41.278
C03092=1015.046,167.855,-134.966,-24.393,21.394,-41.275
C03093=1015.046,168.255,-135.008,-24.393,21.393,-41.273
C03094=1015.044,168.656,-135.051,-24.393,21.393,-41.271
C03095=1015.042,169.056,-135.093,-24.394,21.393,-41.267
C03096=1015.041,169.457,-135.135,-24.394,21.392,-41.265
C03097=1015.039,169.858,-135.177,-24.395,21.392,-41.262
C03098=1015.037,170.258,-135.220,-24.395,21.392,-41.260
C03099=1015.037,170.658,-135.261,-24.395,21.392,-41.256
C03100=1015.035,171.059,-135.304,-24.396,21.392,-41.254
C03101=1015.033,171.459,-135.346,-24.396,21.392,-41.251
C03102=1015.032,171.860,-135.389,-24.396,21.392,-41.249
C03103=1015.031,172.261,-135.431,-24.397,21.391,-41.247
C03104=1015.029,172.661,-135.474,-24.397,21.391,-41.243
C03105=1015.028,173.062,-135.517,-24.397,21.391,-41.242
C03106=1015.026,173.463,-135.559,-24.398,21.390,-41.238
C03107=1015.025,173.862,-135.601,-24.398,21.390,-41.236
C03108=1015.023,174.263,-135.643,-24.399,21.391,-41.233
C03109=1015.022,174.664,-135.686,-24.399,21.390,-41.231
C03110=1015.020,175.065,-135.728,-24.400,21.390,-41.227
C03111=1015.019,175.466,-135.771,-24.400,21.390,-41.225
C03112=1015.018,175.866,-135.813,-24.400,21.390,-41.223
C03113=1015.017,176.267,-135.856,-24.401,21.389,-41.219
C03114=1015.015,176.667,-135.899,-24.401,21.389,-41.218
C03115=1015.014,177.069,-135.941,-24.401,21.389,-41.214
C03116=1015.012,177.469,-135.984,-24.402,21.389,-41.212
C03117=1015.011,177.871,-136.027,-24.402,21.389,-41.209
C03118=1015.010,178.271,-136.070,-24.402,21.388,-41.207
C03119=1015.009,178.672,-136.112,-24.403,21.388,-41.205
C03120=1015.007,179.073,-136.155,-24.403,21.388,-41.201
C03121=1015.006,179.474,-136.198,-24.403,21.388,-41.199
C03122=1015.004,179.874,-136.241,-24.404,21.388,-41.196
C03123=1015.003,180.275,-136.283,-24.404,21.388,-41.194
C03124=1015.002,180.676,-136.326,-24.405,21.387,-41.190
C03125=1015.001,181.077,-136.369,-24.405,21.387,-41.188
C03126=1014.999,181.478,-136.411,-24.405,21.387,-41.186
C03127=1014.998,181.879,-136.454,-24.406,21.387,-41.183
C03128=1014.997,182.280,-136.498,-24.406,21.386,-41.181
C03129=1014.995,182.680,-136.541,-24.407,21.387,-41.177
C03130=1014.994,183.082,-136.583,-24.407,21.386,-41.176
C03131=1014.993,183.483,-136.626,-24.407,21.386,-41.172
C03132=1014.992,183.883,-136.669,-24.408,21.386,-41.170
C03133=1014.991,184.284,-136.712,-24.408,21.386,-41.168
C03134=1014.990,184.685,-136.755,-24.409,21.386,-41.165
C03135=1014.989,185.087,-136.798,-24.409,21.385,-41.162
C03136=1014.987,185.487,-136.841,-24.409,21.385,-41.159
C03137=1014.986,185.888,-136.884,-24.410,21.385,-41.157
C03138=1014.985,186.289,-136.927,-24.410,21.384,-41.155
C03139=1014.984,186.689,-136.970,-24.410,21.384,-41.151
C03140=1014.983,187.091,-137.013,-24.411,21.384,-41.150
C03141=1014.981,187.493,-137.057,-24.411,21.385,-41.146
C03142=1014.980,187.893,-137.100,-24.411,21.384,-41.144
C03143=1014.979,188.294,-137.143,-24.412,21.384,-41.141
C03144=1014.978,188.695,-137.186,-24.412,21.384,-41.139
C03145=1014.977,189.096,-137.229,-24.412,21.384,-41.137
C03146=1014.976,189.497,-137.272,-24.413,21.383,-41.133
C03147=1014.974,189.898,-137.316,-24.413,21.383,-41.131
C03148=1014.973,190.299,-137.359,-24.414,21.383,-41.128
C03149=1014.973,190.701,-137.403,-24.414,21.383,-41.126
C03150=1014.971,191.101,-137.446,-24.414,21.382,-41.124
C03151=1014.971,191.502,-137.489,-24.415,21.382,-41.120
C03152=1014.969,191.904,-137.533,-24.415,21.382,-41.118
C03153=1014.968,192.305,-137.576,-24.415,21.382,-41.115
C03154=1014.967,192.706,-137.619,-24.416,21.382,-41.113
C03155=1014.966,193.107,-137.662,-24.416,21.382,-41.109
C03156=1014.966,193.508,-137.706,-24.417,21.382,-41.108
C03157=1014.964,193.909,-137.750,-24.417,21.381,-41.105
C03158=1014.964,194.310,-137.794,-24.417,21.381,-41.102
C03159=1014.963,194.711,-137.837,-24.418,21.381,-41.100
C03160=1014.962,195.113,-137.880,-24.418,21.381,-41.097
C03161=1014.960,195.513,-137.924,-24.418,21.380,-41.094
C03162=1014.959,195.915,-137.967,-24.419,21.381,-41.091
C03163=1014.959,196.315,-138.011,-24.419,21.380,-41.089
C03164=1014.957,196.717,-138.055,-24.419,21.380,-41.087
C03165=1014.957,197.118,-138.098,-24.420,21.380,-41.084
C03166=1014.956,197.519,-138.142,-24.420,21.380,-41.082
C03167=1014.955,197.920,-138.186,-24.421,21.380,-41.078
C03168=1014.954,198.321,-138.230,-24.421,21.379,-41.076
C03169=1014.953,198.723,-138.273,-24.421,21.379,-41.074
C03170=1014.953,199.121,-138.316,-24.422,21.379,-41.071
C03171=1014.952,199.510,-138.359,-24.422,21.379,-41.069
C03172=1014.951,199.911,-138.403,-24.423,21.378,-41.065
C03173=1014.950,200.123,-138.426,-24.423,21.378,-41.065
C03174=1014.950,200.347,-138.451,-24.423,21.378,-41.063
C03175=1014.950,200.576,-138.475,-24.423,21.378,-41.061
C03176=1014.949,200.802,-138.501,-24.423,21.379,-41.060
C03177=1014.948,201.210,-138.545,-24.424,21.378,-41.058
C03178=1014.948,201.561,-138.583,-24.424,21.378,-41.054
C03179=1014.946,201.911,-138.622,-24.424,21.378,-41.052
C03180=1014.947,202.297,-138.664,-24.425,21.378,-41.051
C03181=1014.952,203.514,-138.800,-24.373,21.403,-41.416
C03182=1014.954,203.761,-138.827,-24.373,21.404,-41.415
C03183=1014.955,204.010,-138.855,-24.373,21.403,-41.414
C03184=1014.957,204.259,-138.882,-24.373,21.403,-41.412
C03185=1014.959,204.507,-138.909,-24.374,21.404,-41.411
C03186=1014.961,204.756,-138.936,-24.373,21.403,-41.410
C03187=1014.963,205.004,-138.964,-24.374,21.403,-41.409
C03188=1014.964,205.253,-138.991,-24.374,21.403,-41.407
C03189=1014.966,205.501,-139.018,-24.374,21.402,-41.407
C03190=1014.968,205.750,-139.046,-24.374,21.403,-41.405
C03191=1014.970,205.998,-139.073,-24.375,21.403,-41.403
C03192=1014.971,206.247,-139.101,-24.375,21.402,-41.401
C03193=1014.973,206.495,-139.128,-24.375,21.402,-41.401
C03194=1014.975,206.744,-139.155,-24.375,21.402,-41.399
C03195=1014.977,206.993,-139.183,-24.375,21.402,-41.398
C03196=1014.979,207.240,-139.211,-24.375,21.402,-41.398
C03197=1014.980,207.489,-139.238,-24.376,21.402,-41.396
C03198=1014.983,207.738,-139.265,-24.376,21.402,-41.394
C03199=1014.984,207.986,-139.293,-24.376,21.402,-41.392
C03200=1014.986,208.229,-139.320,-24.376,21.401,-41.392
C03201=1014.988,208.471,-139.347,-24.376,21.402,-41.391
C03202=1014.990,208.714,-139.373,-24.377,21.402,-41.389
C03203=1014.992,208.957,-139.400,-24.377,21.401,-41.388
C03204=1014.993,209.199,-139.427,-24.377,21.402,-41.387
C03205=1014.995,209.442,-139.454,-24.377,21.401,-41.385
C03206=1014.998,209.685,-139.481,-24.377,21.401,-41.383
C03207=1014.999,209.927,-139.508,-24.377,21.401,-41.383
C03208=1015.001,210.176,-139.535,-24.378,21.401,-41.381
C03209=1015.004,210.424,-139.563,-24.378,21.401,-41.379
C03210=1015.005,210.673,-139.591,-24.378,21.401,-41.378
C03211=1015.007,210.922,-139.618,-24.378,21.400,-41.377
C03212=1015.009,211.169,-139.645,-24.378,21.400,-41.375
C03213=1015.011,211.418,-139.673,-24.379,21.401,-41.374
C03214=1015.013,211.666,-139.701,-24.379,21.401,-41.372
C03215=1015.014,211.915,-139.728,-24.379,21.400,-41.372
C03216=1015.017,212.163,-139.756,-24.379,21.400,-41.370
C03217=1015.019,212.412,-139.784,-24.380,21.400,-41.368
C03218=1015.021,212.660,-139.812,-24.380,21.400,-41.366
C03219=1015.023,212.909,-139.839,-24.380,21.400,-41.366
C03220=1015.025,213.157,-139.867,-24.380,21.400,-41.365
C03221=1015.027,213.405,-139.894,-24.380,21.400,-41.363
C03222=1015.028,213.654,-139.922,-24.381,21.400,-41.361
C03223=1015.031,213.903,-139.950,-24.381,21.400,-41.359
C03224=1015.033,214.151,-139.977,-24.381,21.399,-41.359
C03225=1015.035,214.400,-140.005,-24.381,21.399,-41.357
C03226=1015.037,214.647,-140.033,-24.381,21.400,-41.356
C03227=1015.039,214.897,-140.061,-24.382,21.399,-41.354
C03228=1015.041,215.139,-140.087,-24.382,21.398,-41.353
C03229=1015.043,215.381,-140.115,-24.382,21.399,-41.352
C03230=1015.045,215.624,-140.141,-24.382,21.399,-41.350
C03231=1015.047,215.867,-140.169,-24.382,21.399,-41.348
C03232=1015.049,216.110,-140.196,-24.383,21.398,-41.346
C03233=1015.051,216.352,-140.223,-24.383,21.398,-41.346
C03234=1015.053,216.596,-140.250,-24.383,21.398,-41.344
C03235=1015.055,216.838,-140.277,-24.383,21.398,-41.342
C03236=1015.057,217.086,-140.305,-24.383,21.399,-41.341
C03237=1015.059,217.335,-140.333,-24.384,21.398,-41.339
C03238=1015.062,217.584,-140.361,-24.384,21.397,-41.339
C03239=1015.064,217.832,-140.388,-24.384,21.397,-41.337
C03240=1015.065,218.080,-140.416,-24.384,21.398,-41.335
C03241=1015.068,218.329,-140.444,-24.384,21.398,-41.333
C03242=1015.070,218.577,-140.472,-24.385,21.397,-41.332
C03243=1015.072,218.826,-140.499,-24.385,21.397,-41.330
C03244=1015.074,219.075,-140.528,-24.385,21.397,-41.330
C03245=1015.077,219.322,-140.556,-24.385,21.397,-41.328
C03246=1015.079,219.570,-140.583,-24.385,21.397,-41.326
C03247=1015.081,219.820,-140.611,-24.386,21.397,-41.324
C03248=1015.083,220.068,-140.639,-24.386,21.397,-41.323
C03249=1015.085,220.316,-140.667,-24.386,21.397,-41.321
C03250=1015.088,220.565,-140.695,-24.386,21.396,-41.320
C03251=1015.089,220.813,-140.723,-24.386,21.396,-41.318
C03252=1015.092,221.062,-140.751,-24.387,21.397,-41.317
C03253=1015.094,221.310,-140.779,-24.387,21.396,-41.315
C03254=1015.097,221.559,-140.807,-24.387,21.396,-41.313
C03255=1015.099,221.807,-140.835,-24.388,21.396,-41.311
C03256=1015.101,222.049,-140.862,-24.388,21.397,-41.310
C03257=1015.103,222.292,-140.890,-24.388,21.396,-41.309
C03258=1015.106,222.535,-140.918,-24.388,21.395,-41.308
C03259=1015.108,222.778,-140.944,-24.388,21.395,-41.306
C03260=1015.110,223.021,-140.972,-24.389,21.396,-41.304
C03261=1015.112,223.264,-140.999,-24.389,21.396,-41.302
C03262=1015.114,223.506,-141.026,-24.389,21.395,-41.300
C03263=1015.117,223.750,-141.054,-24.389,21.395,-41.300
C03264=1015.119,223.998,-141.082,-24.389,21.394,-41.298
C03265=1015.121,224.247,-141.111,-24.390,21.395,-41.297
C03266=1015.123,224.494,-141.139,-24.390,21.395,-41.295
C03267=1015.126,224.743,-141.167,-24.390,21.395,-41.293
C03268=1015.128,224.991,-141.195,-24.390,21.394,-41.291
C03269=1015.131,225.240,-141.223,-24.391,21.394,-41.289
C03270=1015.133,225.488,-141.251,-24.391,21.395,-41.288
C03271=1015.136,225.737,-141.279,-24.391,21.395,-41.286
C03272=1015.138,225.985,-141.307,-24.391,21.394,-41.285
C03273=1015.140,226.233,-141.336,-24.391,21.393,-41.284
C03274=1015.142,226.481,-141.363,-24.392,21.393,-41.282
C03275=1015.145,226.730,-141.392,-24.392,21.394,-41.280
C03276=1015.147,226.978,-141.420,-24.392,21.394,-41.278
C03277=1015.149,227.227,-141.448,-24.393,21.393,-41.276
C03278=1015.152,227.476,-141.476,-24.393,21.393,-41.275
C03279=1015.155,227.723,-141.504,-24.393,21.393,-41.273
C03280=1015.157,227.972,-141.533,-24.393,21.394,-41.271
C03281=1015.159,228.220,-141.561,-24.394,21.393,-41.269
C03282=1015.161,228.469,-141.589,-24.394,21.393,-41.267
C03283=1015.164,228.718,-141.617,-24.394,21.393,-41.266
C03284=1015.166,228.961,-141.645,-24.394,21.392,-41.265
C03285=1015.168,229.203,-141.672,-24.394,21.392,-41.263
C03286=1015.172,229.446,-141.700,-24.395,21.392,-41.262
C03287=1015.174,229.689,-141.729,-24.395,21.392,-41.260
C03288=1015.176,229.932,-141.756,-24.395,21.392,-41.258
C03289=1015.179,230.175,-141.783,-24.395,21.392,-41.256
C03290=1015.181,230.418,-141.811,-24.396,21.392,-41.254
C03291=1015.184,230.661,-141.839,-24.396,21.391,-41.252
C03292=1015.186,230.909,-141.868,-24.396,21.392,-41.251
C03293=1015.189,231.157,-141.896,-24.396,21.392,-41.249
C03294=1015.192,231.406,-141.924,-24.397,21.392,-41.247
C03295=1015.193,231.654,-141.952,-24.397,21.391,-41.245
C03296=1015.196,231.903,-141.980,-24.397,21.391,-41.243
C03297=1015.199,232.151,-142.010,-24.397,21.391,-41.242
C03298=1015.202,232.400,-142.038,-24.398,21.391,-41.240
C03299=1015.203,232.648,-142.066,-24.398,21.390,-41.238
C03300=1015.207,232.896,-142.095,-24.398,21.391,-41.236
C03301=1015.210,233.144,-142.123,-24.399,21.391,-41.234
C03302=1015.212,233.393,-142.151,-24.399,21.391,-41.233
C03303=1015.214,233.641,-142.179,-24.399,21.390,-41.231
C03304=1015.217,233.889,-142.209,-24.399,21.390,-41.229
C03305=1015.220,234.138,-142.237,-24.400,21.390,-41.227
C03306=1015.222,234.387,-142.265,-24.400,21.390,-41.225
C03307=1015.224,234.634,-142.294,-24.400,21.390,-41.223
C03308=1015.227,234.883,-142.322,-24.400,21.389,-41.221
C03309=1015.230,235.131,-142.351,-24.401,21.389,-41.219
C03310=1015.233,235.380,-142.379,-24.401,21.389,-41.218
C03311=1015.235,235.628,-142.408,-24.401,21.390,-41.216
C03312=1015.238,235.871,-142.436,-24.401,21.389,-41.214
C03313=1015.240,236.114,-142.464,-24.402,21.389,-41.212
C03314=1015.243,236.357,-142.491,-24.402,21.389,-41.210
C03315=1015.245,236.600,-142.520,-24.402,21.389,-41.209
C03316=1015.248,236.843,-142.548,-24.402,21.388,-41.207
C03317=1015.251,237.087,-142.576,-24.403,21.388,-41.205
C03318=1015.254,237.329,-142.604,-24.403,21.388,-41.203
C03319=1015.256,237.572,-142.632,-24.403,21.388,-41.201
C03320=1015.259,237.820,-142.661,-24.403,21.388,-41.199
C03321=1015.262,238.069,-142.689,-24.404,21.387,-41.197
C03322=1015.264,238.317,-142.718,-24.404,21.387,-41.195
C03323=1015.267,238.566,-142.746,-24.405,21.388,-41.192
C03324=1015.270,238.814,-142.776,-24.405,21.387,-41.190
C03325=1015.273,239.063,-142.804,-24.405,21.387,-41.188
C03326=1015.275,239.311,-142.833,-24.405,21.387,-41.186
C03327=1015.278,239.559,-142.861,-24.406,21.387,-41.184
C03328=1015.282,239.807,-142.890,-24.406,21.386,-41.183
C03329=1015.284,240.056,-142.919,-24.406,21.386,-41.181
C03330=1015.287,240.304,-142.948,-24.406,21.386,-41.179
C03331=1015.290,240.553,-142.977,-24.407,21.386,-41.177
C03332=1015.293,240.801,-143.006,-24.407,21.386,-41.174
C03333=1015.295,241.049,-143.034,-24.407,21.386,-41.172
C03334=1015.298,241.297,-143.063,-24.408,21.386,-41.170
C03335=1015.301,241.546,-143.092,-24.408,21.386,-41.168
C03336=1015.303,241.782,-143.120,-24.408,21.385,-41.166
C03337=1015.306,242.019,-143.147,-24.408,21.385,-41.164
C03338=1015.309,242.255,-143.175,-24.409,21.385,-41.162
C03339=1015.312,242.492,-143.202,-24.409,21.385,-41.160
C03340=1015.314,242.728,-143.229,-24.409,21.384,-41.159
C03341=1015.317,242.966,-143.257,-24.410,21.385,-41.155
C03342=1015.320,243.202,-143.285,-24.410,21.385,-41.153
C03343=1015.323,243.439,-143.312,-24.410,21.384,-41.151
C03344=1015.325,243.700,-143.343,-24.411,21.384,-41.150
C03345=1015.329,243.962,-143.373,-24.411,21.384,-41.148
C03346=1015.332,244.223,-143.403,-24.411,21.384,-41.146
C03347=1015.335,244.484,-143.434,-24.412,21.384,-41.143
C03348=1015.338,244.732,-143.463,-24.412,21.384,-41.141
C03349=1015.340,244.981,-143.492,-24.412,21.384,-41.139
C03350=1015.343,245.229,-143.520,-24.412,21.384,-41.137
C03351=1015.346,245.477,-143.550,-24.413,21.384,-41.134
C03352=1015.350,245.726,-143.579,-24.413,21.384,-41.132
C03353=1015.353,245.974,-143.608,-24.413,21.383,-41.129
C03354=1015.356,246.222,-143.637,-24.414,21.382,-41.127
C03355=1015.359,246.470,-143.666,-24.414,21.382,-41.126
C03356=1015.361,246.718,-143.695,-24.414,21.383,-41.122
C03357=1015.365,246.966,-143.724,-24.415,21.382,-41.120
C03358=1015.368,247.215,-143.754,-24.415,21.382,-41.118
C03359=1015.371,247.463,-143.782,-24.415,21.382,-41.117
C03360=1015.374,247.712,-143.812,-24.416,21.382,-41.113
C03361=1015.377,247.960,-143.841,-24.416,21.382,-41.111
C03362=1015.379,248.208,-143.870,-24.416,21.381,-41.109
C03363=1015.383,248.457,-143.899,-24.417,21.381,-41.107
C03364=1015.386,248.705,-143.929,-24.417,21.381,-41.104
C03365=1015.389,248.953,-143.957,-24.417,21.381,-41.102
C03366=1015.392,249.201,-143.987,-24.418,21.381,-41.100
C03367=1015.395,249.450,-144.016,-24.418,21.381,-41.098
C03368=1015.398,249.693,-144.045,-24.418,21.381,-41.095
C03369=1015.401,249.937,-144.073,-24.419,21.381,-41.093
C03370=1015.404,250.180,-144.102,-24.419,21.380,-41.091
C03371=1015.407,250.423,-144.131,-24.419,21.380,-41.089
C03372=1015.410,250.666,-144.159,-24.420,21.380,-41.085
C03373=1015.414,250.909,-144.188,-24.420,21.380,-41.084
C03374=1015.416,251.153,-144.216,-24.420,21.380,-41.082
C03375=1015.420,251.396,-144.245,-24.421,21.380,-41.078
C03376=1015.422,251.645,-144.274,-24.421,21.380,-41.076
C03377=1015.426,251.892,-144.304,-24.421,21.379,-41.074
C03378=1015.429,252.141,-144.334,-24.421,21.378,-41.072
C03379=1015.432,252.389,-144.362,-24.422,21.379,-41.069
C03380=1015.435,252.637,-144.392,-24.422,21.379,-41.067
C03381=1015.439,252.886,-144.421,-24.423,21.378,-41.065
C03382=1015.441,253.133,-144.451,-24.423,21.378,-41.061
C03383=1015.445,253.382,-144.480,-24.423,21.378,-41.060
C03384=1015.448,253.630,-144.510,-24.424,21.378,-41.058
C03385=1015.451,253.878,-144.539,-24.424,21.378,-41.054
C03386=1015.454,254.127,-144.569,-24.424,21.378,-41.052
C03387=1015.458,254.375,-144.598,-24.425,21.377,-41.049
C03388=1015.461,254.624,-144.627,-24.425,21.377,-41.047
C03389=1015.464,254.871,-144.657,-24.425,21.377,-41.045
C03390=1015.467,255.119,-144.686,-24.426,21.377,-41.042
C03391=1015.470,255.368,-144.716,-24.426,21.377,-41.040
C03392=1015.474,255.616,-144.745,-24.426,21.376,-41.037
C03393=1015.477,255.865,-144.775,-24.427,21.376,-41.034
C03394=1015.480,256.112,-144.805,-24.427,21.376,-41.032
C03395=1015.483,256.361,-144.834,-24.428,21.377,-41.029
C03396=1015.487,256.604,-144.863,-24.428,21.376,-41.027
C03397=1015.490,256.848,-144.892,-24.428,21.375,-41.025
C03398=1015.493,257.091,-144.921,-24.429,21.376,-41.021
C03399=1015.496,257.335,-144.950,-24.429,21.376,-41.019
C03400=1015.500,257.578,-144.979,-24.429,21.375,-41.018
C03401=1015.503,257.821,-145.008,-24.430,21.375,-41.014
C03402=1015.506,258.065,-145.038,-24.430,21.375,-41.012
C03403=1015.522,259.301,-145.190,-24.551,21.322,-40.171
C03404=1015.525,259.580,-145.226,-24.587,21.310,-39.930
C03405=1015.527,259.860,-145.264,-24.622,21.298,-39.688
C03406=1015.528,260.139,-145.302,-24.658,21.287,-39.446
C03407=1015.529,260.418,-145.339,-24.693,21.275,-39.204
C03408=1015.530,260.666,-145.374,-24.725,21.267,-38.988
C03409=1015.530,260.914,-145.409,-24.758,21.259,-38.770
C03410=1015.530,261.162,-145.444,-24.790,21.251,-38.554
C03411=1015.529,261.408,-145.479,-24.823,21.245,-38.337
C03412=1015.528,261.688,-145.521,-24.860,21.238,-38.090
C03413=1015.526,261.967,-145.563,-24.897,21.233,-37.842
C03414=1015.525,262.247,-145.606,-24.935,21.227,-37.593
C03415=1015.522,262.526,-145.649,-24.973,21.223,-37.345
C03416=1015.520,262.773,-145.688,-25.006,21.220,-37.124
C03417=1015.517,263.020,-145.727,-25.040,21.217,-36.903
C03418=1015.513,263.267,-145.767,-25.074,21.216,-36.681
C03419=1015.511,263.514,-145.807,-25.108,21.215,-36.458
C03420=1015.506,263.793,-145.854,-25.147,21.216,-36.205
C03421=1015.500,264.072,-145.900,-25.186,21.217,-35.952
C03422=1015.496,264.351,-145.948,-25.226,21.219,-35.699
C03423=1015.491,264.630,-145.997,-25.265,21.221,-35.444
C03424=1015.484,264.876,-146.040,-25.300,21.225,-35.219
C03425=1015.478,265.122,-146.083,-25.335,21.229,-34.991
C03426=1015.472,265.368,-146.127,-25.370,21.233,-34.766
C03427=1015.466,265.614,-146.172,-25.406,21.239,-34.538
C03428=1015.457,265.893,-146.223,-25.446,21.246,-34.279
C03429=1015.449,266.172,-146.275,-25.487,21.254,-34.021
C03430=1015.441,266.451,-146.328,-25.527,21.264,-33.760
C03431=1015.432,266.729,-146.381,-25.568,21.275,-33.499
C03432=1015.423,266.974,-146.428,-25.604,21.284,-33.268
C03433=1015.414,267.220,-146.477,-25.641,21.295,-33.037
C03434=1015.405,267.465,-146.526,-25.677,21.306,-32.805
C03435=1015.395,267.710,-146.575,-25.714,21.319,-32.571
C03436=1015.383,267.989,-146.631,-25.755,21.334,-32.305
C03437=1015.372,268.267,-146.688,-25.797,21.350,-32.039
C03438=1015.360,268.547,-146.746,-25.839,21.367,-31.772
C03439=1015.347,268.824,-146.805,-25.881,21.386,-31.502
C03440=1015.335,269.069,-146.856,-25.918,21.402,-31.266
C03441=1015.323,269.313,-146.908,-25.955,21.420,-31.029
C03442=1015.310,269.557,-146.962,-25.992,21.438,-30.791
C03443=1015.297,269.801,-147.015,-26.030,21.459,-30.551
C03444=1015.283,270.079,-147.076,-26.072,21.483,-30.277
C03445=1015.267,270.358,-147.139,-26.115,21.507,-30.003
C03446=1015.251,270.636,-147.202,-26.158,21.533,-29.728
C03447=1015.235,270.914,-147.266,-26.201,21.560,-29.450
C03448=1015.220,271.158,-147.322,-26.238,21.585,-29.208
C03449=1015.205,271.400,-147.378,-26.276,21.610,-28.964
C03450=1015.189,271.643,-147.436,-26.314,21.637,-28.720
C03451=1015.174,271.886,-147.493,-26.351,21.664,-28.476
C03452=1015.155,272.164,-147.561,-26.395,21.697,-28.194
C03453=1015.136,272.442,-147.628,-26.438,21.731,-27.910
C03454=1015.116,272.720,-147.696,-26.481,21.766,-27.626
C03455=1015.097,272.998,-147.765,-26.525,21.803,-27.342
C03456=1015.079,273.240,-147.826,-26.562,21.835,-27.092
C03457=1015.061,273.482,-147.887,-26.600,21.869,-26.841
C03458=1015.042,273.724,-147.948,-26.638,21.904,-26.589
C03459=1015.022,273.965,-148.011,-26.676,21.940,-26.336
C03460=1015.000,274.243,-148.083,-26.720,21.983,-26.043
C03461=1014.977,274.520,-148.157,-26.763,22.027,-25.750
C03462=1014.953,274.798,-148.230,-26.807,22.073,-25.453
C03463=1014.930,275.075,-148.304,-26.851,22.119,-25.156
C03464=1014.909,275.316,-148.369,-26.889,22.162,-24.896
C03465=1014.888,275.556,-148.435,-26.927,22.204,-24.635
C03466=1014.866,275.797,-148.502,-26.965,22.250,-24.373
C03467=1014.843,276.037,-148.569,-27.003,22.295,-24.109
C03468=1014.817,276.314,-148.646,-27.046,22.349,-23.804
C03469=1014.790,276.591,-148.725,-27.090,22.404,-23.496
C03470=1014.763,276.868,-148.804,-27.134,22.462,-23.186
C03471=1014.736,277.145,-148.884,-27.177,22.521,-22.877
C03472=1014.711,277.384,-148.954,-27.215,22.573,-22.606
C03473=1014.687,277.622,-149.024,-27.252,22.626,-22.334
C03474=1014.661,277.861,-149.094,-27.290,22.681,-22.062
C03475=1014.636,278.100,-149.166,-27.327,22.737,-21.789
C03476=1014.606,278.376,-149.249,-27.370,22.804,-21.469
C03477=1014.575,278.653,-149.333,-27.413,22.872,-21.148
C03478=1014.544,278.929,-149.418,-27.456,22.942,-20.824
C03479=1014.512,279.206,-149.504,-27.498,23.014,-20.499
C03480=1014.484,279.443,-149.579,-27.534,23.078,-20.218
C03481=1014.456,279.680,-149.654,-27.570,23.143,-19.936
C03482=1014.427,279.917,-149.729,-27.606,23.208,-19.653
C03483=1014.398,280.154,-149.805,-27.642,23.276,-19.367
C03484=1014.364,280.429,-149.893,-27.684,23.357,-19.031
C03485=1014.329,280.705,-149.984,-27.725,23.440,-18.691
C03486=1014.295,280.982,-150.075,-27.766,23.526,-18.349
C03487=1014.259,281.257,-150.167,-27.807,23.613,-18.004
C03488=1014.227,281.491,-150.245,-27.842,23.690,-17.706
C03489=1014.196,281.727,-150.325,-27.877,23.768,-17.406
C03490=1014.163,281.962,-150.405,-27.911,23.848,-17.104
C03491=1014.131,282.197,-150.486,-27.945,23.929,-16.801
C03492=1014.093,282.472,-150.582,-27.984,24.027,-16.441
C03493=1014.053,282.747,-150.677,-28.023,24.128,-16.079
C03494=1014.014,283.022,-150.775,-28.062,24.232,-15.713
C03495=1013.974,283.297,-150.872,-28.100,24.338,-15.343
C03496=1013.939,283.528,-150.956,-28.132,24.429,-15.026
C03497=1013.904,283.762,-151.041,-28.164,24.524,-14.708
C03498=1013.869,283.995,-151.126,-28.195,24.619,-14.388
C03499=1013.833,284.227,-151.211,-28.226,24.716,-14.065
C03500=1013.790,284.501,-151.313,-28.261,24.835,-13.680
C03501=1013.746,284.775,-151.416,-28.296,24.955,-13.292
C03502=1013.702,285.049,-151.518,-28.330,25.079,-12.901
C03503=1013.657,285.322,-151.623,-28.364,25.204,-12.507
C03504=1013.619,285.553,-151.712,-28.391,25.314,-12.171
C03505=1013.580,285.783,-151.801,-28.418,25.425,-11.832
C03506=1013.541,286.013,-151.891,-28.444,25.537,-11.492
C03507=1013.501,286.243,-151.982,-28.470,25.652,-11.148
C03508=1013.453,286.516,-152.090,-28.499,25.792,-10.737
C03509=1013.405,286.788,-152.200,-28.527,25.936,-10.320
C03510=1013.356,287.061,-152.309,-28.555,26.082,-9.899
C03511=1013.306,287.332,-152.421,-28.581,26.233,-9.471
C03512=1013.264,287.561,-152.515,-28.602,26.363,-9.109
C03513=1013.222,287.788,-152.609,-28.622,26.495,-8.743
C03514=1013.179,288.015,-152.704,-28.641,26.630,-8.372
C03515=1013.135,288.243,-152.801,-28.659,26.767,-7.999
C03516=1013.082,288.513,-152.916,-28.679,26.937,-7.545
C03517=1013.029,288.784,-153.032,-28.698,27.109,-7.088
C03518=1012.975,289.055,-153.149,-28.715,27.285,-6.624
C03519=1012.921,289.325,-153.267,-28.730,27.467,-6.153
C03520=1012.875,289.550,-153.366,-28.742,27.622,-5.757
C03521=1012.828,289.775,-153.466,-28.752,27.779,-5.357
C03522=1012.781,289.999,-153.567,-28.760,27.939,-4.952
C03523=1012.734,290.223,-153.668,-28.767,28.103,-4.544
C03524=1012.676,290.492,-153.791,-28.773,28.305,-4.046
C03525=1012.617,290.761,-153.914,-28.777,28.512,-3.541
C03526=1012.557,291.029,-154.039,-28.778,28.722,-3.030
C03527=1012.497,291.297,-154.165,-28.777,28.937,-2.514
C03528=1012.447,291.518,-154.270,-28.773,29.120,-2.080
C03529=1012.397,291.740,-154.376,-28.768,29.306,-1.642
C03530=1012.345,291.960,-154.482,-28.760,29.495,-1.198
C03531=1012.293,292.181,-154.589,-28.751,29.688,-0.751
C03532=1012.230,292.447,-154.720,-28.736,29.926,-0.203
C03533=1012.166,292.713,-154.851,-28.717,30.168,0.353
C03534=1012.101,292.979,-154.984,-28.695,30.417,0.916
C03535=1012.035,293.244,-155.117,-28.669,30.673,1.490
C03536=1011.980,293.462,-155.228,-28.645,30.886,1.967
C03537=1011.925,293.678,-155.340,-28.617,31.104,2.450
C03538=1011.869,293.895,-155.452,-28.586,31.327,2.940
C03539=1011.813,294.112,-155.564,-28.552,31.552,3.436
C03540=1011.744,294.376,-155.704,-28.506,31.835,4.050
C03541=1011.674,294.639,-155.843,-28.455,32.122,4.672
C03542=1011.602,294.902,-155.985,-28.398,32.417,5.306
C03543=1011.531,295.163,-156.127,-28.335,32.716,5.947
C03544=1011.471,295.376,-156.244,-28.280,32.966,6.479
C03545=1011.412,295.589,-156.362,-28.220,33.220,7.016
C03546=1011.351,295.801,-156.480,-28.156,33.478,7.560
C03547=1011.290,296.013,-156.599,-28.087,33.739,8.111
C03548=1011.214,296.274,-156.746,-27.996,34.069,8.801
C03549=1011.138,296.534,-156.895,-27.897,34.404,9.500
C03550=1011.061,296.792,-157.046,-27.790,34.746,10.213
C03551=1010.982,297.050,-157.197,-27.675,35.094,10.935
C03552=1010.918,297.259,-157.320,-27.576,35.380,11.529
C03553=1010.854,297.466,-157.444,-27.470,35.670,12.129
C03554=1010.789,297.674,-157.569,-27.359,35.965,12.738
C03555=1010.723,297.879,-157.694,-27.241,36.263,13.354
C03556=1010.640,298.136,-157.851,-27.085,36.641,14.134
C03557=1010.557,298.392,-158.009,-26.918,37.024,14.926
C03558=1010.472,298.647,-158.169,-26.741,37.414,15.733
C03559=1010.387,298.901,-158.330,-26.551,37.810,16.553
C03560=1010.319,299.103,-158.459,-26.391,38.132,17.220
C03561=1010.249,299.305,-158.589,-26.221,38.458,17.898
C03562=1010.179,299.507,-158.721,-26.044,38.788,18.586
C03563=1010.108,299.708,-158.853,-25.857,39.121,19.283
///RCONF 0,0,0,0,0,0,0,0,0,0,0,0,0,0,0,0,0,0,0,0,0,0,0,0
C03564=1010.018,299.959,-159.020,-25.611,39.544,20.170
C03565=1009.928,300.210,-159.188,-25.349,39.974,21.077
C03566=1009.836,300.459,-159.357,-25.071,40.409,21.999
C03567=1009.744,300.708,-159.528,-24.778,40.847,22.938
C03568=1009.670,300.904,-159.663,-24.533,41.199,23.695
C03569=1009.595,301.100,-159.801,-24.278,41.553,24.463
C03570=1009.520,301.296,-159.939,-24.010,41.911,25.245
C03571=1009.444,301.490,-160.077,-23.731,42.271,26.037
C03572=1009.347,301.736,-160.253,-23.359,42.732,27.060
C03573=1009.249,301.981,-160.431,-22.967,43.196,28.105
C03574=1009.150,302.225,-160.611,-22.552,43.665,29.173
C03575=1009.051,302.468,-160.792,-22.115,44.137,30.264
C03576=1008.971,302.658,-160.935,-21.757,44.508,31.133
C03577=1008.892,302.846,-161.078,-21.384,44.880,32.017
C03578=1008.811,303.035,-161.223,-20.996,45.254,32.916
C03579=1008.730,303.222,-161.367,-20.592,45.628,33.828
